// TIA Portal project "SistemaSupervisorio" (V17)
// Engenharia de Software 1

(* hardware
DEVICE "S7-1500/ET200MP station_1"  S7-1500 station
   slot 0: "RACK_CPU_1500"  Rack  6ES7 590-1***0-0AA0
   slot 1: "CPU_1500"  CPU 1511-1 PN  6ES7 511-1AK00-0AB0  V1.8
      slot 3: "CPU display_1"  6ES7591-1AA00-0AA0
      slot 32768: "PROFINET interface_1500"  X1
         slot 32769: "Port_1"  X1 P1
         slot 32770: "Port_2"  X1 P2
   slot 2: "DI1_1500"  DI 16x24VDC BA  6ES7 521-1BH10-0AA0  V1.1
   slot 3: "DO1_1500"  DQ 16x24VDC/0.5A BA  6ES7 522-1BH10-0AA0  V1.1
   slot 4: "AI/AO1_1500"  AI/AQ 4xU/I/RTD/TC / 2xU/I ST  6ES7 534-7QE00-0AB0  V1.0
*)

// ===== PLC "CPU_1500"  CPU 1511-1 PN =====

VAR_GLOBAL   // PLC tag table "Default tag table"
   "%I0.0" AT %I0.0 : Bool;   // I0.0 - Channel0 InDigitalCPU_1500
   "%I0.1" AT %I0.1 : Bool;   // I0.1 - Channel1 InDigitalCPU_1500
   "%I0.2" AT %I0.2 : Bool;   // I0.2 - Channel2 InDigitalCPU_1500
   "%I0.3" AT %I0.3 : Bool;   // I0.3 - Channel3 InDigitalCPU_1500
   "%I0.4" AT %I0.4 : Bool;   // I0.4 - Channel4 InDigitalCPU_1500
   "%I0.5" AT %I0.5 : Bool;   // I0.5 - Channel5 InDigitalCPU_1500
   "%I0.6" AT %I0.6 : Bool;   // I0.6 - Channel6 InDigitalCPU_1500
   "%I0.7" AT %I0.7 : Bool;   // I0.7 - Channel7 InDigitalCPU_1500
   "%I1.0" AT %I1.0 : Bool;   // I1.0 - Channel10 InDigitalCPU_1500
   "%I1.1" AT %I1.1 : Bool;   // I1.1 - Channel11 InDigitalCPU_1500
   "%I1.2" AT %I1.2 : Bool;   // I1.2 - Channel12 InDigitalCPU_1500
   "%I1.3" AT %I1.3 : Bool;   // I1.3 - Channel13 InDigitalCPU_1500
   "%I1.4" AT %I1.4 : Bool;   // I1.4 - Channel14 InDigitalCPU_1500
   "%I1.5" AT %I1.5 : Bool;   // I1.5 - Channel15 InDigitalCPU_1500
   "%I1.6" AT %I1.6 : Bool;   // I1.6 - Channel16 InDigitalCPU_1500
   "%I1.7" AT %I1.7 : Bool;   // I1.7 - Channel17 InDigitalCPU_1500
   "%IW2" AT %IW2 : Int;   // IW2 - Channel0 InAnalogAI/AO_1500
   "%IW4" AT %IW4 : Int;   // IW4 - Channel1 InAnalogAI/AO_1500
   "%IW6" AT %IW6 : Int;   // IW6 - Channel3 InAnalogAI/AO_1500
   "%IW8" AT %IW8 : Int;   // IW8 - Channel4 InAnalogAI/AO_1500
   "%QW2" AT %QW2 : Int;   // %QW2 - Channel0 OutAnalogAI/AO_1500
   "%QW4" AT %QW4 : Int;   // %QW4 - Channel1 OutAnalogAI/AO_1500
   "%Q0.0" AT %Q0.0 : Bool;   // Q0.0 - Channel0 OutDigitalDO_1500
   "%Q0.1" AT %Q0.1 : Bool;   // Q0.1 - Channel1 OutDigitalDO_1500
   "%Q0.2" AT %Q0.2 : Bool;   // Q1.0 - Channel2 OutDigitalDO_1500
   "%Q0.3" AT %Q0.3 : Bool;   // Q0.3 - Channel3 OutDigitalDO_1500
   "%Q0.4" AT %Q0.4 : Bool;   // Q0.4 - Channel4 OutDigitalDO_1500
   "%Q0.5" AT %Q0.5 : Bool;   // Q0.5 - Channel5 OutDigitalDO_1500
   "%Q0.6" AT %Q0.6 : Bool;   // Q0.6 - Channel6 OutDigitalDO_1500
   "%Q0.7" AT %Q0.7 : Bool;   // Q0.7 - Channel7 OutDigitalDO_1500
   "%Q1.0" AT %Q1.0 : Bool;   // Q1.0 - Channel10 OutDigitalDO_1500
   "%Q1.1" AT %Q1.1 : Bool;   // Q1.1 - Channel11 OutDigitalDO_1500
   "%Q1.2" AT %Q1.2 : Bool;   // Q1.2 - Channel12 OutDigitalDO_1500
   "%Q1.3" AT %Q1.3 : Bool;   // Q1.3 - Channel13 OutDigitalDO_1500
   "%Q1.4" AT %Q1.4 : Bool;   // Q1.4 - Channel14 OutDigitalDO_1500
   "%Q1.5" AT %Q1.5 : Bool;   // Q1.5 - Channel15 OutDigitalDO_1500
   "%Q1.6" AT %Q1.6 : Bool;   // Q1.6 - Channel16 OutDigitalDO_1500
   "%Q1.7" AT %Q1.7 : Bool;   // Q1.7 - Channel17 OutDigitalDO_1500
   "System_Byte" AT %MB100 : Byte;
   "FirstScan" AT %M100.0 : Bool;
   "DiagStatusUpdate" AT %M100.1 : Bool;
   "AlwaysTRUE" AT %M100.2 : Bool;
   "AlwaysFALSE" AT %M100.3 : Bool;
   "Tag_1" AT %M150.1 : Bool;
END_VAR

// folder: 001 - IOs/DBs

DATA_BLOCK "Ed"   // DB1
{ S7_Optimized_Access := 'FALSE' }
VERSION : 0.1
   VAR
      "I0.0" : Bool;   // I0.0 - Channel0 InDigitalCPU_ENG1
      "I0.1" : Bool;   // I0.1 - Channel1 InDigitalCPU_ENG1
      "I0.2" : Bool;   // I0.2 - Channel2 InDigitalCPU_ENG1
      "I0.3" : Bool;   // I0.3 - Channel3 InDigitalCPU_ENG1
      "I0.4" : Bool;   // I0.4 - Channel4 InDigitalCPU_ENG1
      "I0.5" : Bool;   // I0.5 - Channel5 InDigitalCPU_ENG1
      "I0.6" : Bool;   // I0.6 - Channel6 InDigitalCPU_ENG1
      "I0.7" : Bool;   // I0.7 - Channel7 InDigitalCPU_ENG1
      "I1.0" : Bool;   // I1.0 - Channel8 InDigitalCPU_ENG1
      "I1.1" : Bool;   // I1.1 - Channel9 InDigitalCPU_ENG1
      "I1.2" : Bool;   // I1.2 - Channel10, InDigitalCPU_ENG1
      "I1.3" : Bool;   // I1.3 - Channel11 InDigitalCPU_ENG1
      "I1.4" : Bool;   // I1.4 - Channel12 InDigitalCPU_ENG1
      "I1.5" : Bool;   // I1.5 - Channel13 InDigitalCPU_ENG1
      "I1.6" : Bool;
      "I1.7" : Bool;
      Simulation : Struct
         Ed : Struct
            "I0.0" : Bool;
            "I0.1" : Bool;
            "I0.2" : Bool;
            "I0.3" : Bool;
            "I0.4" : Bool;
            "I0.5" : Bool;
            "I0.6" : Bool;
            "I0.7" : Bool;
            "I1.0" : Bool;
            "I1.1" : Bool;
            "I1.2" : Bool;
            "I1.3" : Bool;
            "I1.4" : Bool;
            "I1.5" : Bool;
            "I1.6" : Bool;
            "I1.7" : Bool;
         END_STRUCT;
         Test : Struct
            "I0.0" : Bool;
            "I0.1" : Bool;
            "I0.2" : Bool;
            "I0.3" : Bool;
            "I0.4" : Bool;
            "I0.5" : Bool;
            "I0.6" : Bool;
            "I0.7" : Bool;
            "I1.0" : Bool;
            "I1.1" : Bool;
            "I1.2" : Bool;
            "I1.3" : Bool;
            "I1.4" : Bool;
            "I1.5" : Bool;
            "I1.6" : Bool;
            "I1.7" : Bool;
            All : Bool;
         END_STRUCT;
         Enable : Struct
            "I0.0" : Bool;
            "I0.1" : Bool;
            "I0.2" : Bool;
            "I0.3" : Bool;
            "I0.4" : Bool;
            "I0.5" : Bool;
            "I0.6" : Bool;
            "I0.7" : Bool;
            "I1.0" : Bool;
            "I1.1" : Bool;
            "I1.2" : Bool;
            "I1.3" : Bool;
            "I1.4" : Bool;
            "I1.5" : Bool;
            "I1.6" : Bool;
            "I1.7" : Bool;
            All : Bool;
         END_STRUCT;
      END_STRUCT;
   END_VAR
BEGIN
END_DATA_BLOCK

DATA_BLOCK "Sd"   // DB2
{ S7_Optimized_Access := 'FALSE' }
VERSION : 0.1
   VAR
      "Q0.0" : Bool;   // Q0.0 - Channel0 OutDigitalCPU_ENG1
      "Q0.1" : Bool;   // Q0.1 - Channel1 OutDigitalCPU_ENG1
      "Q0.2" : Bool;   // Q0.2 - Channel2 OutDigitalCPU_ENG1
      "Q0.3" : Bool;   // Q0.3 - Channel3 OutDigitalCPU_ENG1
      "Q0.4" : Bool;   // Q0.4 - Channel4 OutDigitalCPU_ENG1
      "Q0.5" : Bool;   // Q0.5 - Channel5 OutDigitalCPU_ENG1
      "Q0.6" : Bool;   // Q0.6 - Channel6 OutDigitalCPU_ENG1
      "Q0.7" : Bool;   // Q0.7 - Channel7 OutDigitalCPU_ENG1
      "Q1.0" : Bool;   // Q1.1 - Channel8 OutDigitalCPU_ENG1
      "Q1.1" : Bool;   // Q1.2 - Channel9 OutDigitalCPU_ENG1
      "Q1.2" : Bool;
      "Q1.3" : Bool;
      "Q1.4" : Bool;
      "Q1.5" : Bool;
      "Q1.6" : Bool;
      "Q1.7" : Bool;
      Simulation : Struct
         Sd : Struct
            "Q0.0" : Bool;   // Q0.0 - Channel0 OutDigitalCPU_ENG1
            "Q0.1" : Bool;   // Q0.1 - Channel1 OutDigitalCPU_ENG1
            "Q0.2" : Bool;   // Q0.2 - Channel2 OutDigitalCPU_ENG1
            "Q0.3" : Bool;   // Q0.3 - Channel3 OutDigitalCPU_ENG1
            "Q0.4" : Bool;   // Q0.4 - Channel4 OutDigitalCPU_ENG1
            "Q0.5" : Bool;   // Q0.5 - Channel5 OutDigitalCPU_ENG1
            "Q0.6" : Bool;   // Q0.6 - Channel6 OutDigitalCPU_ENG1
            "Q0.7" : Bool;   // Q0.7 - Channel7 OutDigitalCPU_ENG1
            "Q1.0" : Bool;   // Q1.1 - Channel8 OutDigitalCPU_ENG1
            "Q1.1" : Bool;   // Q1.2 - Channel9 OutDigitalCPU_ENG1
            "Q1.2" : Bool;
            "Q1.3" : Bool;
            "Q1.4" : Bool;
            "Q1.5" : Bool;
            "Q1.6" : Bool;
            "Q1.7" : Bool;
         END_STRUCT;
         Test : Struct
            "Q0.0" : Bool;
            "Q0.1" : Bool;
            "Q0.2" : Bool;
            "Q0.3" : Bool;
            "Q0.4" : Bool;
            "Q0.5" : Bool;
            "Q0.6" : Bool;
            "Q0.7" : Bool;
            "Q1.0" : Bool;
            "Q1.1" : Bool;
            "Q1.2" : Bool;
            "Q1.3" : Bool;
            "Q1.4" : Bool;
            "Q1.5" : Bool;
            "Q1.6" : Bool;
            "Q1.7" : Bool;
            All : Bool;
         END_STRUCT;
         Enable : Struct
            "Q0.0" : Bool;
            "Q0.1" : Bool;
            "Q0.2" : Bool;
            "Q0.3" : Bool;
            "Q0.4" : Bool;
            "Q0.5" : Bool;
            "Q0.6" : Bool;
            "Q0.7" : Bool;
            "Q1.0" : Bool;
            "Q1.1" : Bool;
            "Q1.2" : Bool;
            "Q1.3" : Bool;
            "Q1.4" : Bool;
            "Q1.5" : Bool;
            "Q1.6" : Bool;
            "Q1.7" : Bool;
            All : Bool;
         END_STRUCT;
      END_STRUCT;
   END_VAR
BEGIN
END_DATA_BLOCK

DATA_BLOCK "Ea"   // DB3
{ S7_Optimized_Access := 'FALSE' }
VERSION : 0.1
   VAR
      IW2 : Int;   // IW64 - Channel0 InAnalogCPU_ENG1
      IW4 : Int;   // IW66 - Channel1 InAnalogCPU_ENG1
      IW6 : Int;   // IW96 - Channel0 InAnalogAI/AO_ENG1
      IW8 : Int;   // IW98 - Channel1 InAnalogAI/AO_ENG1
      Simulation : Struct
         Ea : Struct
            IW2 : Int;   // IW64 - Channel0 InAnalogCPU_ENG1
            IW4 : Int;   // IW66 - Channel1 InAnalogCPU_ENG1
            IW6 : Int;   // IW96 - Channel0 InAnalogAI/AO_ENG1
            IW8 : Int;   // IW98 - Channel1 InAnalogAI/AO_ENG1
         END_STRUCT;
         Test : Struct
            IW2 : DInt;   // IW64 - Channel0 InAnalogCPU_ENG1
            IW4 : DInt;   // IW66 - Channel1 InAnalogCPU_ENG1
            IW6 : DInt;   // IW96 - Channel0 InAnalogAI/AO_ENG1
            IW8 : DInt;   // IW98 - Channel1 InAnalogAI/AO_ENG1
            All : DInt;
         END_STRUCT;
         Enable : Struct
            IW2 : Bool;   // IW64 - Channel0 InAnalogCPU_ENG1
            IW4 : Bool;   // IW66 - Channel1 InAnalogCPU_ENG1
            IW6 : Bool;   // IW96 - Channel0 InAnalogAI/AO_ENG1
            IW8 : Bool;   // IW98 - Channel1 InAnalogAI/AO_ENG1
            All : Bool;
         END_STRUCT;
      END_STRUCT;
   END_VAR
BEGIN
END_DATA_BLOCK

DATA_BLOCK "Sa"   // DB4
{ S7_Optimized_Access := 'FALSE' }
VERSION : 0.1
   VAR
      QW2 : Int;   // IW96 - Channel0 OutAnalogCPU_AI/AO
      QW4 : Int;   // IW98 - Channel1 OutAnalogCPU_AI/AO
      Simulation : Struct
         Sa : Struct
            QW2 : Int;
            QW4 : Int;
         END_STRUCT;
         Test : Struct
            QW2 : DInt;
            QW4 : DInt;
            All : DInt;
         END_STRUCT;
         Enable : Struct
            QW2 : Bool;
            QW4 : Bool;
            All : Bool;
         END_STRUCT;
      END_STRUCT;
   END_VAR
BEGIN
END_DATA_BLOCK

// folder: 002 - Comunication Node-Red/DBs

DATA_BLOCK "Node-Red"   // DB6
{ S7_Optimized_Access := 'FALSE' }
VERSION : 0.1
   VAR
      escreveNodeRedBool : Bool;
      escreveNodeRedDint : DInt;
      recebeNodeRedBool : Bool;
      recebeNodeRedReal : Real;
      auxEscreveNodRedReal : DInt;
      auxRecebeNodeRedReal : DInt;
      statusMaquinaNodeRed : Int;
      "enviaStatusNode-Red" : Int;
      avisosMaquinaNodeRed : Int;
      enviaAvisosMaquinaNodeRed : Int;
      "alarmesNode-Red" : Int;
      enviaAlarmesNodeRed : Int;
      "valorVelocidadeNode-Red" : Int;
      "enviaValorVelocidadeNode-Red" : Int;
      valorProducao : Int;
      enviaValorProducao : Int;
      enableEnviaValorProdução : Bool;
      enableEnviaValorVelocidade : Bool;
   END_VAR
BEGIN
END_DATA_BLOCK

// folder: 100 - DBs

DATA_BLOCK "x"   // DB5
{ S7_Optimized_Access := 'TRUE' }
VERSION : 0.1
   VAR RETAIN
      Constantes : Struct
         "+int" : Int := 32767;
         "-int" : Int := -32767;
         "0int" : Int := 0;
      END_STRUCT;
      AlwaysFalse : Bool := 0;
      AlwaysTrue : Bool := 1;
   END_VAR
   VAR
      Timers : Struct
         t1s : Bool;
         t5s : Bool;
         t10s : Bool;
      END_STRUCT;
   END_VAR
BEGIN
END_DATA_BLOCK

// folder: System blocks/Program resources

DATA_BLOCK "tonTimer5seg"   // DB7
{ S7_Optimized_Access := 'TRUE' }
AUTHOR : Simatic
FAMILY : IEC
NAME : IEC_TMR
VERSION : 1.0
// stored: InstanceOfName IEC_TIMER
"IEC_TIMER"
BEGIN
END_DATA_BLOCK

DATA_BLOCK "tonTimer10seg"   // DB8
{ S7_Optimized_Access := 'TRUE' }
AUTHOR : Simatic
FAMILY : IEC
NAME : IEC_TMR
VERSION : 1.0
// stored: InstanceOfName IEC_TIMER
"IEC_TIMER"
BEGIN
END_DATA_BLOCK

DATA_BLOCK "tonTimer1seg"   // DB9
{ S7_Optimized_Access := 'TRUE' }
AUTHOR : Simatic
FAMILY : IEC
NAME : IEC_TMR
VERSION : 1.0
// stored: InstanceOfName IEC_TIMER
"IEC_TIMER"
BEGIN
END_DATA_BLOCK

// folder: (top level)

ORGANIZATION_BLOCK "Main"   // OB1, LAD, ProgramCycle
TITLE = "Main Program Sweep (Cycle)"
{ S7_Optimized_Access := 'TRUE' }
VERSION : 0.1
   VAR_INPUT
      Initial_Call : Bool;   // Initial call of this OB
      Remanence : Bool;   // =True, if remanent data are available
   END_VAR
BEGIN

REGION Network 1: 01 - Digital Inputs
   // 01 - Digital Input
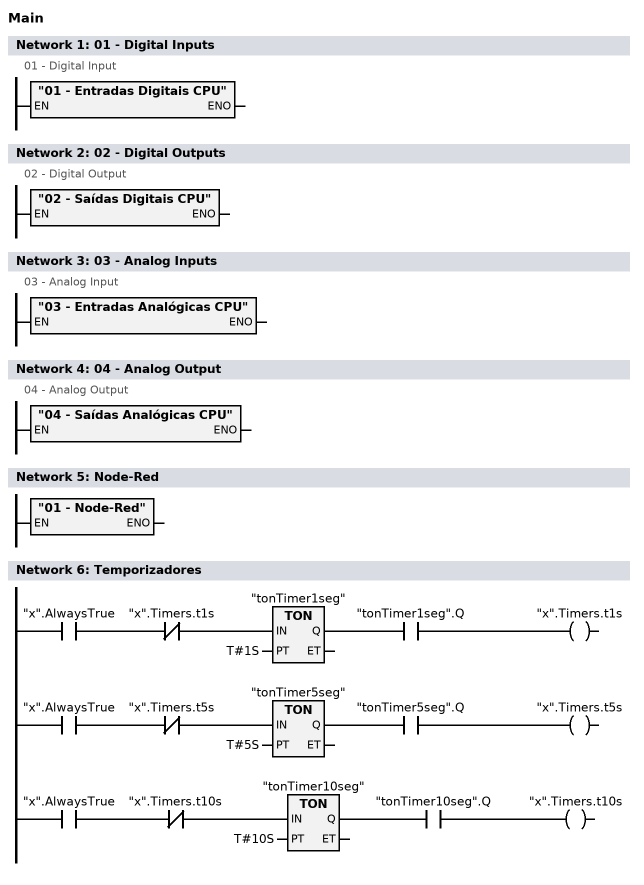
   RUNG wire#powerrail
      "01 - Entradas Digitais CPU"()
   END_RUNG
   // the same network as SCL:
   "01 - Entradas Digitais CPU"();
END_REGION

REGION Network 2: 02 - Digital Outputs
   // 02 - Digital Output
   RUNG wire#powerrail
      "02 - Saídas Digitais CPU"()
   END_RUNG
   // the same network as SCL:
   "02 - Saídas Digitais CPU"();
END_REGION

REGION Network 3: 03 - Analog Inputs
   // 03 - Analog Input
   RUNG wire#powerrail
      "03 - Entradas Analógicas CPU"()
   END_RUNG
   // the same network as SCL:
   "03 - Entradas Analógicas CPU"();
END_REGION

REGION Network 4: 04 - Analog Output
   // 04 - Analog Output
   RUNG wire#powerrail
      "04 - Saídas Analógicas CPU"()
   END_RUNG
   // the same network as SCL:
   "04 - Saídas Analógicas CPU"();
END_REGION

REGION Network 5: Node-Red
   RUNG wire#powerrail
      "01 - Node-Red"()
   END_RUNG
   // the same network as SCL:
   "01 - Node-Red"();
END_REGION

REGION Network 6: Temporizadores
   "tonTimer1seg".TON(IN := "x".AlwaysTrue AND NOT "x".Timers.t1s, PT := T#1S);
   "x".Timers.t1s := "tonTimer1seg".Q AND "tonTimer1seg".Q;
   "tonTimer5seg".TON(IN := "x".AlwaysTrue AND NOT "x".Timers.t5s, PT := T#5S);
   "x".Timers.t5s := "tonTimer5seg".Q AND "tonTimer5seg".Q;
   "tonTimer10seg".TON(IN := "x".AlwaysTrue AND NOT "x".Timers.t10s, PT := T#10S);
   "x".Timers.t10s := "tonTimer10seg".Q AND "tonTimer10seg".Q;
END_REGION
END_ORGANIZATION_BLOCK

// folder: 001 - IOs

FUNCTION "01 - Entradas Digitais CPU" : Void   // FC1, LAD
TITLE = 01 - Digital Inputs
{ S7_Optimized_Access := 'TRUE' }
VERSION : 0.1
// 01 - Digital Inputs
   VAR_TEMP
      testeAllHabilitado : Bool;
      testeAllDesabilitado : Bool;
   END_VAR
BEGIN

REGION Network 1: 00 - Digital Input %I0.0
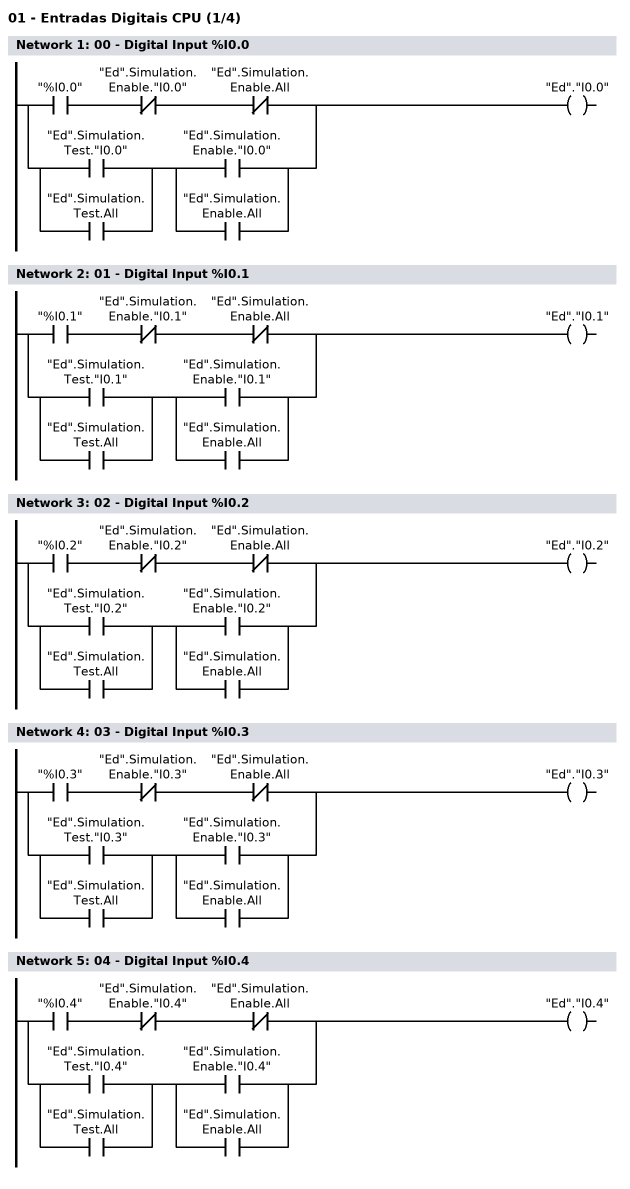
   RUNG wire#powerrail
      Contact( "%I0.0" )
      I_Contact( "Ed".Simulation.Enable."I0.0" )
      I_Contact( "Ed".Simulation.Enable.All )
      wire#w1
      Coil( "Ed"."I0.0" )
   END_RUNG
   RUNG wire#powerrail
      Contact( "Ed".Simulation.Test."I0.0" )
      wire#w2
      Contact( "Ed".Simulation.Enable."I0.0" )
   END_RUNG wire#w1
   RUNG wire#powerrail
      Contact( "Ed".Simulation.Test.All )
   END_RUNG wire#w2
   RUNG wire#w2
      Contact( "Ed".Simulation.Enable.All )
   END_RUNG wire#w1
   // the same network as SCL:
   "Ed"."I0.0" := ("%I0.0" AND NOT "Ed".Simulation.Enable."I0.0" AND NOT "Ed".Simulation.Enable.All) OR (("Ed".Simulation.Test."I0.0" OR "Ed".Simulation.Test.All) AND ("Ed".Simulation.Enable."I0.0" OR "Ed".Simulation.Enable.All));
END_REGION

REGION Network 2: 01 - Digital Input %I0.1
   RUNG wire#powerrail
      Contact( "%I0.1" )
      I_Contact( "Ed".Simulation.Enable."I0.1" )
      I_Contact( "Ed".Simulation.Enable.All )
      wire#w1
      Coil( "Ed"."I0.1" )
   END_RUNG
   RUNG wire#powerrail
      Contact( "Ed".Simulation.Test."I0.1" )
      wire#w2
      Contact( "Ed".Simulation.Enable."I0.1" )
   END_RUNG wire#w1
   RUNG wire#powerrail
      Contact( "Ed".Simulation.Test.All )
   END_RUNG wire#w2
   RUNG wire#w2
      Contact( "Ed".Simulation.Enable.All )
   END_RUNG wire#w1
   // the same network as SCL:
   "Ed"."I0.1" := ("%I0.1" AND NOT "Ed".Simulation.Enable."I0.1" AND NOT "Ed".Simulation.Enable.All) OR (("Ed".Simulation.Test."I0.1" OR "Ed".Simulation.Test.All) AND ("Ed".Simulation.Enable."I0.1" OR "Ed".Simulation.Enable.All));
END_REGION

REGION Network 3: 02 - Digital Input %I0.2
   RUNG wire#powerrail
      Contact( "%I0.2" )
      I_Contact( "Ed".Simulation.Enable."I0.2" )
      I_Contact( "Ed".Simulation.Enable.All )
      wire#w1
      Coil( "Ed"."I0.2" )
   END_RUNG
   RUNG wire#powerrail
      Contact( "Ed".Simulation.Test."I0.2" )
      wire#w2
      Contact( "Ed".Simulation.Enable."I0.2" )
   END_RUNG wire#w1
   RUNG wire#powerrail
      Contact( "Ed".Simulation.Test.All )
   END_RUNG wire#w2
   RUNG wire#w2
      Contact( "Ed".Simulation.Enable.All )
   END_RUNG wire#w1
   // the same network as SCL:
   "Ed"."I0.2" := ("%I0.2" AND NOT "Ed".Simulation.Enable."I0.2" AND NOT "Ed".Simulation.Enable.All) OR (("Ed".Simulation.Test."I0.2" OR "Ed".Simulation.Test.All) AND ("Ed".Simulation.Enable."I0.2" OR "Ed".Simulation.Enable.All));
END_REGION

REGION Network 4: 03 - Digital Input %I0.3
   RUNG wire#powerrail
      Contact( "%I0.3" )
      I_Contact( "Ed".Simulation.Enable."I0.3" )
      I_Contact( "Ed".Simulation.Enable.All )
      wire#w1
      Coil( "Ed"."I0.3" )
   END_RUNG
   RUNG wire#powerrail
      Contact( "Ed".Simulation.Test."I0.3" )
      wire#w2
      Contact( "Ed".Simulation.Enable."I0.3" )
   END_RUNG wire#w1
   RUNG wire#powerrail
      Contact( "Ed".Simulation.Test.All )
   END_RUNG wire#w2
   RUNG wire#w2
      Contact( "Ed".Simulation.Enable.All )
   END_RUNG wire#w1
   // the same network as SCL:
   "Ed"."I0.3" := ("%I0.3" AND NOT "Ed".Simulation.Enable."I0.3" AND NOT "Ed".Simulation.Enable.All) OR (("Ed".Simulation.Test."I0.3" OR "Ed".Simulation.Test.All) AND ("Ed".Simulation.Enable."I0.3" OR "Ed".Simulation.Enable.All));
END_REGION

REGION Network 5: 04 - Digital Input %I0.4
   RUNG wire#powerrail
      Contact( "%I0.4" )
      I_Contact( "Ed".Simulation.Enable."I0.4" )
      I_Contact( "Ed".Simulation.Enable.All )
      wire#w1
      Coil( "Ed"."I0.4" )
   END_RUNG
   RUNG wire#powerrail
      Contact( "Ed".Simulation.Test."I0.4" )
      wire#w2
      Contact( "Ed".Simulation.Enable."I0.4" )
   END_RUNG wire#w1
   RUNG wire#powerrail
      Contact( "Ed".Simulation.Test.All )
   END_RUNG wire#w2
   RUNG wire#w2
      Contact( "Ed".Simulation.Enable.All )
   END_RUNG wire#w1
   // the same network as SCL:
   "Ed"."I0.4" := ("%I0.4" AND NOT "Ed".Simulation.Enable."I0.4" AND NOT "Ed".Simulation.Enable.All) OR (("Ed".Simulation.Test."I0.4" OR "Ed".Simulation.Test.All) AND ("Ed".Simulation.Enable."I0.4" OR "Ed".Simulation.Enable.All));
END_REGION

REGION Network 6: 05 - Digital Input %I0.5
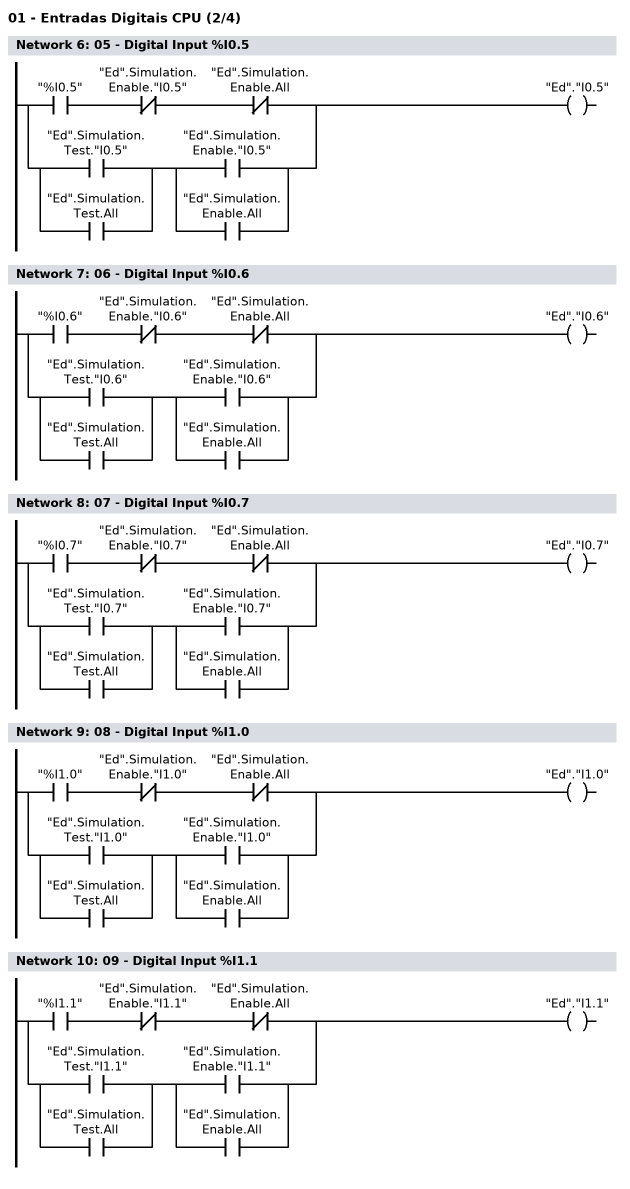
   RUNG wire#powerrail
      Contact( "%I0.5" )
      I_Contact( "Ed".Simulation.Enable."I0.5" )
      I_Contact( "Ed".Simulation.Enable.All )
      wire#w1
      Coil( "Ed"."I0.5" )
   END_RUNG
   RUNG wire#powerrail
      Contact( "Ed".Simulation.Test."I0.5" )
      wire#w2
      Contact( "Ed".Simulation.Enable."I0.5" )
   END_RUNG wire#w1
   RUNG wire#powerrail
      Contact( "Ed".Simulation.Test.All )
   END_RUNG wire#w2
   RUNG wire#w2
      Contact( "Ed".Simulation.Enable.All )
   END_RUNG wire#w1
   // the same network as SCL:
   "Ed"."I0.5" := ("%I0.5" AND NOT "Ed".Simulation.Enable."I0.5" AND NOT "Ed".Simulation.Enable.All) OR (("Ed".Simulation.Test."I0.5" OR "Ed".Simulation.Test.All) AND ("Ed".Simulation.Enable."I0.5" OR "Ed".Simulation.Enable.All));
END_REGION

REGION Network 7: 06 - Digital Input %I0.6
   RUNG wire#powerrail
      Contact( "%I0.6" )
      I_Contact( "Ed".Simulation.Enable."I0.6" )
      I_Contact( "Ed".Simulation.Enable.All )
      wire#w1
      Coil( "Ed"."I0.6" )
   END_RUNG
   RUNG wire#powerrail
      Contact( "Ed".Simulation.Test."I0.6" )
      wire#w2
      Contact( "Ed".Simulation.Enable."I0.6" )
   END_RUNG wire#w1
   RUNG wire#powerrail
      Contact( "Ed".Simulation.Test.All )
   END_RUNG wire#w2
   RUNG wire#w2
      Contact( "Ed".Simulation.Enable.All )
   END_RUNG wire#w1
   // the same network as SCL:
   "Ed"."I0.6" := ("%I0.6" AND NOT "Ed".Simulation.Enable."I0.6" AND NOT "Ed".Simulation.Enable.All) OR (("Ed".Simulation.Test."I0.6" OR "Ed".Simulation.Test.All) AND ("Ed".Simulation.Enable."I0.6" OR "Ed".Simulation.Enable.All));
END_REGION

REGION Network 8: 07 - Digital Input %I0.7
   RUNG wire#powerrail
      Contact( "%I0.7" )
      I_Contact( "Ed".Simulation.Enable."I0.7" )
      I_Contact( "Ed".Simulation.Enable.All )
      wire#w1
      Coil( "Ed"."I0.7" )
   END_RUNG
   RUNG wire#powerrail
      Contact( "Ed".Simulation.Test."I0.7" )
      wire#w2
      Contact( "Ed".Simulation.Enable."I0.7" )
   END_RUNG wire#w1
   RUNG wire#powerrail
      Contact( "Ed".Simulation.Test.All )
   END_RUNG wire#w2
   RUNG wire#w2
      Contact( "Ed".Simulation.Enable.All )
   END_RUNG wire#w1
   // the same network as SCL:
   "Ed"."I0.7" := ("%I0.7" AND NOT "Ed".Simulation.Enable."I0.7" AND NOT "Ed".Simulation.Enable.All) OR (("Ed".Simulation.Test."I0.7" OR "Ed".Simulation.Test.All) AND ("Ed".Simulation.Enable."I0.7" OR "Ed".Simulation.Enable.All));
END_REGION

REGION Network 9: 08 - Digital Input %I1.0
   RUNG wire#powerrail
      Contact( "%I1.0" )
      I_Contact( "Ed".Simulation.Enable."I1.0" )
      I_Contact( "Ed".Simulation.Enable.All )
      wire#w1
      Coil( "Ed"."I1.0" )
   END_RUNG
   RUNG wire#powerrail
      Contact( "Ed".Simulation.Test."I1.0" )
      wire#w2
      Contact( "Ed".Simulation.Enable."I1.0" )
   END_RUNG wire#w1
   RUNG wire#powerrail
      Contact( "Ed".Simulation.Test.All )
   END_RUNG wire#w2
   RUNG wire#w2
      Contact( "Ed".Simulation.Enable.All )
   END_RUNG wire#w1
   // the same network as SCL:
   "Ed"."I1.0" := ("%I1.0" AND NOT "Ed".Simulation.Enable."I1.0" AND NOT "Ed".Simulation.Enable.All) OR (("Ed".Simulation.Test."I1.0" OR "Ed".Simulation.Test.All) AND ("Ed".Simulation.Enable."I1.0" OR "Ed".Simulation.Enable.All));
END_REGION

REGION Network 10: 09 - Digital Input %I1.1
   RUNG wire#powerrail
      Contact( "%I1.1" )
      I_Contact( "Ed".Simulation.Enable."I1.1" )
      I_Contact( "Ed".Simulation.Enable.All )
      wire#w1
      Coil( "Ed"."I1.1" )
   END_RUNG
   RUNG wire#powerrail
      Contact( "Ed".Simulation.Test."I1.1" )
      wire#w2
      Contact( "Ed".Simulation.Enable."I1.1" )
   END_RUNG wire#w1
   RUNG wire#powerrail
      Contact( "Ed".Simulation.Test.All )
   END_RUNG wire#w2
   RUNG wire#w2
      Contact( "Ed".Simulation.Enable.All )
   END_RUNG wire#w1
   // the same network as SCL:
   "Ed"."I1.1" := ("%I1.1" AND NOT "Ed".Simulation.Enable."I1.1" AND NOT "Ed".Simulation.Enable.All) OR (("Ed".Simulation.Test."I1.1" OR "Ed".Simulation.Test.All) AND ("Ed".Simulation.Enable."I1.1" OR "Ed".Simulation.Enable.All));
END_REGION

REGION Network 11: 10 - Digital Input %I1.2
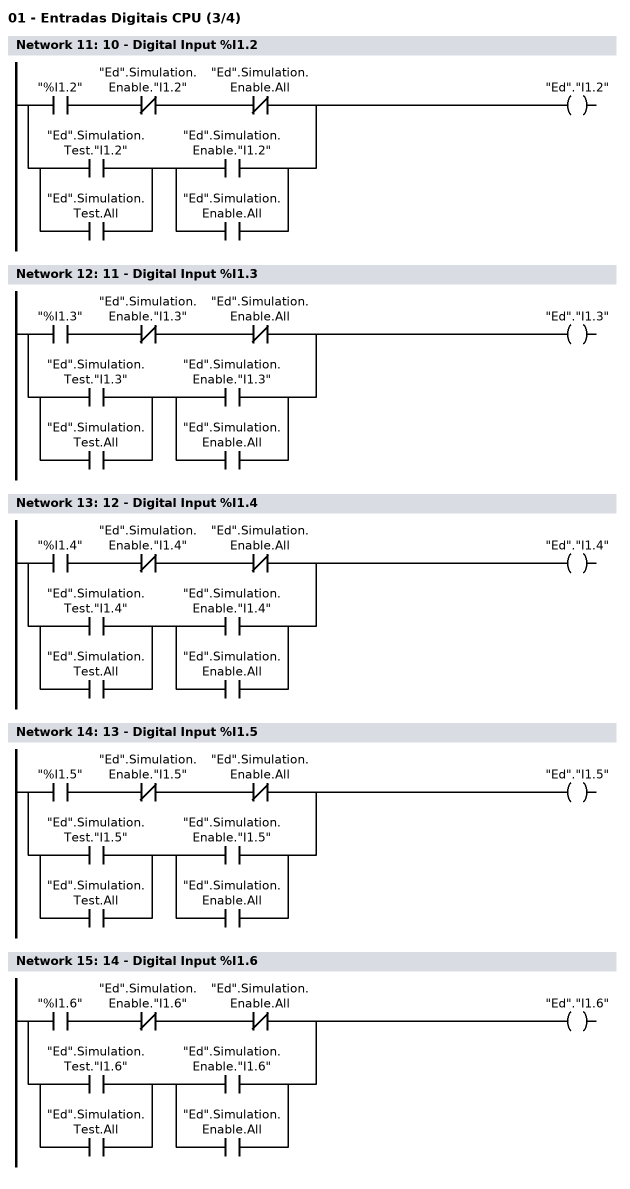
   RUNG wire#powerrail
      Contact( "%I1.2" )
      I_Contact( "Ed".Simulation.Enable."I1.2" )
      I_Contact( "Ed".Simulation.Enable.All )
      wire#w1
      Coil( "Ed"."I1.2" )
   END_RUNG
   RUNG wire#powerrail
      Contact( "Ed".Simulation.Test."I1.2" )
      wire#w2
      Contact( "Ed".Simulation.Enable."I1.2" )
   END_RUNG wire#w1
   RUNG wire#powerrail
      Contact( "Ed".Simulation.Test.All )
   END_RUNG wire#w2
   RUNG wire#w2
      Contact( "Ed".Simulation.Enable.All )
   END_RUNG wire#w1
   // the same network as SCL:
   "Ed"."I1.2" := ("%I1.2" AND NOT "Ed".Simulation.Enable."I1.2" AND NOT "Ed".Simulation.Enable.All) OR (("Ed".Simulation.Test."I1.2" OR "Ed".Simulation.Test.All) AND ("Ed".Simulation.Enable."I1.2" OR "Ed".Simulation.Enable.All));
END_REGION

REGION Network 12: 11 - Digital Input %I1.3
   RUNG wire#powerrail
      Contact( "%I1.3" )
      I_Contact( "Ed".Simulation.Enable."I1.3" )
      I_Contact( "Ed".Simulation.Enable.All )
      wire#w1
      Coil( "Ed"."I1.3" )
   END_RUNG
   RUNG wire#powerrail
      Contact( "Ed".Simulation.Test."I1.3" )
      wire#w2
      Contact( "Ed".Simulation.Enable."I1.3" )
   END_RUNG wire#w1
   RUNG wire#powerrail
      Contact( "Ed".Simulation.Test.All )
   END_RUNG wire#w2
   RUNG wire#w2
      Contact( "Ed".Simulation.Enable.All )
   END_RUNG wire#w1
   // the same network as SCL:
   "Ed"."I1.3" := ("%I1.3" AND NOT "Ed".Simulation.Enable."I1.3" AND NOT "Ed".Simulation.Enable.All) OR (("Ed".Simulation.Test."I1.3" OR "Ed".Simulation.Test.All) AND ("Ed".Simulation.Enable."I1.3" OR "Ed".Simulation.Enable.All));
END_REGION

REGION Network 13: 12 - Digital Input %I1.4
   RUNG wire#powerrail
      Contact( "%I1.4" )
      I_Contact( "Ed".Simulation.Enable."I1.4" )
      I_Contact( "Ed".Simulation.Enable.All )
      wire#w1
      Coil( "Ed"."I1.4" )
   END_RUNG
   RUNG wire#powerrail
      Contact( "Ed".Simulation.Test."I1.4" )
      wire#w2
      Contact( "Ed".Simulation.Enable."I1.4" )
   END_RUNG wire#w1
   RUNG wire#powerrail
      Contact( "Ed".Simulation.Test.All )
   END_RUNG wire#w2
   RUNG wire#w2
      Contact( "Ed".Simulation.Enable.All )
   END_RUNG wire#w1
   // the same network as SCL:
   "Ed"."I1.4" := ("%I1.4" AND NOT "Ed".Simulation.Enable."I1.4" AND NOT "Ed".Simulation.Enable.All) OR (("Ed".Simulation.Test."I1.4" OR "Ed".Simulation.Test.All) AND ("Ed".Simulation.Enable."I1.4" OR "Ed".Simulation.Enable.All));
END_REGION

REGION Network 14: 13 - Digital Input %I1.5
   RUNG wire#powerrail
      Contact( "%I1.5" )
      I_Contact( "Ed".Simulation.Enable."I1.5" )
      I_Contact( "Ed".Simulation.Enable.All )
      wire#w1
      Coil( "Ed"."I1.5" )
   END_RUNG
   RUNG wire#powerrail
      Contact( "Ed".Simulation.Test."I1.5" )
      wire#w2
      Contact( "Ed".Simulation.Enable."I1.5" )
   END_RUNG wire#w1
   RUNG wire#powerrail
      Contact( "Ed".Simulation.Test.All )
   END_RUNG wire#w2
   RUNG wire#w2
      Contact( "Ed".Simulation.Enable.All )
   END_RUNG wire#w1
   // the same network as SCL:
   "Ed"."I1.5" := ("%I1.5" AND NOT "Ed".Simulation.Enable."I1.5" AND NOT "Ed".Simulation.Enable.All) OR (("Ed".Simulation.Test."I1.5" OR "Ed".Simulation.Test.All) AND ("Ed".Simulation.Enable."I1.5" OR "Ed".Simulation.Enable.All));
END_REGION

REGION Network 15: 14 - Digital Input %I1.6
   RUNG wire#powerrail
      Contact( "%I1.6" )
      I_Contact( "Ed".Simulation.Enable."I1.6" )
      I_Contact( "Ed".Simulation.Enable.All )
      wire#w1
      Coil( "Ed"."I1.6" )
   END_RUNG
   RUNG wire#powerrail
      Contact( "Ed".Simulation.Test."I1.6" )
      wire#w2
      Contact( "Ed".Simulation.Enable."I1.6" )
   END_RUNG wire#w1
   RUNG wire#powerrail
      Contact( "Ed".Simulation.Test.All )
   END_RUNG wire#w2
   RUNG wire#w2
      Contact( "Ed".Simulation.Enable.All )
   END_RUNG wire#w1
   // the same network as SCL:
   "Ed"."I1.6" := ("%I1.6" AND NOT "Ed".Simulation.Enable."I1.6" AND NOT "Ed".Simulation.Enable.All) OR (("Ed".Simulation.Test."I1.6" OR "Ed".Simulation.Test.All) AND ("Ed".Simulation.Enable."I1.6" OR "Ed".Simulation.Enable.All));
END_REGION

REGION Network 16: 15 - Digital Input %I1.7
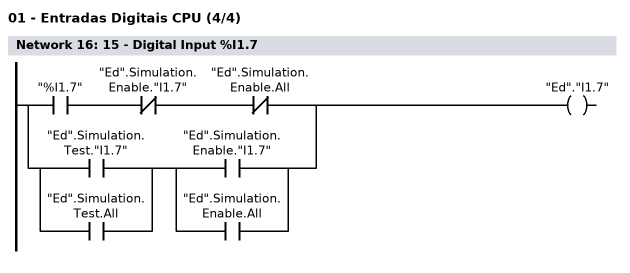
   RUNG wire#powerrail
      Contact( "%I1.7" )
      I_Contact( "Ed".Simulation.Enable."I1.7" )
      I_Contact( "Ed".Simulation.Enable.All )
      wire#w1
      Coil( "Ed"."I1.7" )
   END_RUNG
   RUNG wire#powerrail
      Contact( "Ed".Simulation.Test."I1.7" )
      wire#w2
      Contact( "Ed".Simulation.Enable."I1.7" )
   END_RUNG wire#w1
   RUNG wire#powerrail
      Contact( "Ed".Simulation.Test.All )
   END_RUNG wire#w2
   RUNG wire#w2
      Contact( "Ed".Simulation.Enable.All )
   END_RUNG wire#w1
   // the same network as SCL:
   "Ed"."I1.7" := ("%I1.7" AND NOT "Ed".Simulation.Enable."I1.7" AND NOT "Ed".Simulation.Enable.All) OR (("Ed".Simulation.Test."I1.7" OR "Ed".Simulation.Test.All) AND ("Ed".Simulation.Enable."I1.7" OR "Ed".Simulation.Enable.All));
END_REGION
END_FUNCTION

FUNCTION "02 - Saídas Digitais CPU" : Void   // FC2, LAD
TITLE = 01 - Digital Outputs
{ S7_Optimized_Access := 'TRUE' }
VERSION : 0.1
// 01 - Digital Outputs
BEGIN

REGION Network 1: 02 - Digital Output %Q0.0
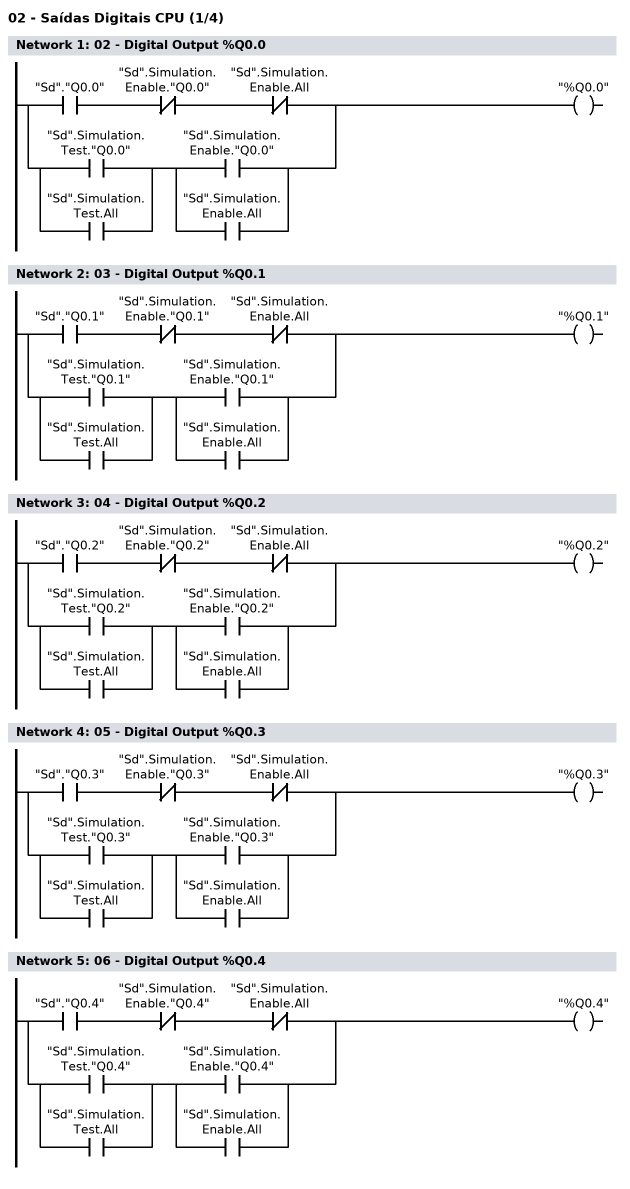
   RUNG wire#powerrail
      Contact( "Sd"."Q0.0" )
      I_Contact( "Sd".Simulation.Enable."Q0.0" )
      I_Contact( "Sd".Simulation.Enable.All )
      wire#w1
      Coil( "%Q0.0" )
   END_RUNG
   RUNG wire#powerrail
      Contact( "Sd".Simulation.Test."Q0.0" )
      wire#w2
      Contact( "Sd".Simulation.Enable."Q0.0" )
   END_RUNG wire#w1
   RUNG wire#powerrail
      Contact( "Sd".Simulation.Test.All )
   END_RUNG wire#w2
   RUNG wire#w2
      Contact( "Sd".Simulation.Enable.All )
   END_RUNG wire#w1
   // the same network as SCL:
   "%Q0.0" := ("Sd"."Q0.0" AND NOT "Sd".Simulation.Enable."Q0.0" AND NOT "Sd".Simulation.Enable.All) OR (("Sd".Simulation.Test."Q0.0" OR "Sd".Simulation.Test.All) AND ("Sd".Simulation.Enable."Q0.0" OR "Sd".Simulation.Enable.All));
END_REGION

REGION Network 2: 03 - Digital Output %Q0.1
   RUNG wire#powerrail
      Contact( "Sd"."Q0.1" )
      I_Contact( "Sd".Simulation.Enable."Q0.1" )
      I_Contact( "Sd".Simulation.Enable.All )
      wire#w1
      Coil( "%Q0.1" )
   END_RUNG
   RUNG wire#powerrail
      Contact( "Sd".Simulation.Test."Q0.1" )
      wire#w2
      Contact( "Sd".Simulation.Enable."Q0.1" )
   END_RUNG wire#w1
   RUNG wire#powerrail
      Contact( "Sd".Simulation.Test.All )
   END_RUNG wire#w2
   RUNG wire#w2
      Contact( "Sd".Simulation.Enable.All )
   END_RUNG wire#w1
   // the same network as SCL:
   "%Q0.1" := ("Sd"."Q0.1" AND NOT "Sd".Simulation.Enable."Q0.1" AND NOT "Sd".Simulation.Enable.All) OR (("Sd".Simulation.Test."Q0.1" OR "Sd".Simulation.Test.All) AND ("Sd".Simulation.Enable."Q0.1" OR "Sd".Simulation.Enable.All));
END_REGION

REGION Network 3: 04 - Digital Output %Q0.2
   RUNG wire#powerrail
      Contact( "Sd"."Q0.2" )
      I_Contact( "Sd".Simulation.Enable."Q0.2" )
      I_Contact( "Sd".Simulation.Enable.All )
      wire#w1
      Coil( "%Q0.2" )
   END_RUNG
   RUNG wire#powerrail
      Contact( "Sd".Simulation.Test."Q0.2" )
      wire#w2
      Contact( "Sd".Simulation.Enable."Q0.2" )
   END_RUNG wire#w1
   RUNG wire#powerrail
      Contact( "Sd".Simulation.Test.All )
   END_RUNG wire#w2
   RUNG wire#w2
      Contact( "Sd".Simulation.Enable.All )
   END_RUNG wire#w1
   // the same network as SCL:
   "%Q0.2" := ("Sd"."Q0.2" AND NOT "Sd".Simulation.Enable."Q0.2" AND NOT "Sd".Simulation.Enable.All) OR (("Sd".Simulation.Test."Q0.2" OR "Sd".Simulation.Test.All) AND ("Sd".Simulation.Enable."Q0.2" OR "Sd".Simulation.Enable.All));
END_REGION

REGION Network 4: 05 - Digital Output %Q0.3
   RUNG wire#powerrail
      Contact( "Sd"."Q0.3" )
      I_Contact( "Sd".Simulation.Enable."Q0.3" )
      I_Contact( "Sd".Simulation.Enable.All )
      wire#w1
      Coil( "%Q0.3" )
   END_RUNG
   RUNG wire#powerrail
      Contact( "Sd".Simulation.Test."Q0.3" )
      wire#w2
      Contact( "Sd".Simulation.Enable."Q0.3" )
   END_RUNG wire#w1
   RUNG wire#powerrail
      Contact( "Sd".Simulation.Test.All )
   END_RUNG wire#w2
   RUNG wire#w2
      Contact( "Sd".Simulation.Enable.All )
   END_RUNG wire#w1
   // the same network as SCL:
   "%Q0.3" := ("Sd"."Q0.3" AND NOT "Sd".Simulation.Enable."Q0.3" AND NOT "Sd".Simulation.Enable.All) OR (("Sd".Simulation.Test."Q0.3" OR "Sd".Simulation.Test.All) AND ("Sd".Simulation.Enable."Q0.3" OR "Sd".Simulation.Enable.All));
END_REGION

REGION Network 5: 06 - Digital Output %Q0.4
   RUNG wire#powerrail
      Contact( "Sd"."Q0.4" )
      I_Contact( "Sd".Simulation.Enable."Q0.4" )
      I_Contact( "Sd".Simulation.Enable.All )
      wire#w1
      Coil( "%Q0.4" )
   END_RUNG
   RUNG wire#powerrail
      Contact( "Sd".Simulation.Test."Q0.4" )
      wire#w2
      Contact( "Sd".Simulation.Enable."Q0.4" )
   END_RUNG wire#w1
   RUNG wire#powerrail
      Contact( "Sd".Simulation.Test.All )
   END_RUNG wire#w2
   RUNG wire#w2
      Contact( "Sd".Simulation.Enable.All )
   END_RUNG wire#w1
   // the same network as SCL:
   "%Q0.4" := ("Sd"."Q0.4" AND NOT "Sd".Simulation.Enable."Q0.4" AND NOT "Sd".Simulation.Enable.All) OR (("Sd".Simulation.Test."Q0.4" OR "Sd".Simulation.Test.All) AND ("Sd".Simulation.Enable."Q0.4" OR "Sd".Simulation.Enable.All));
END_REGION

REGION Network 6: 07 - Digital Output %Q0.5
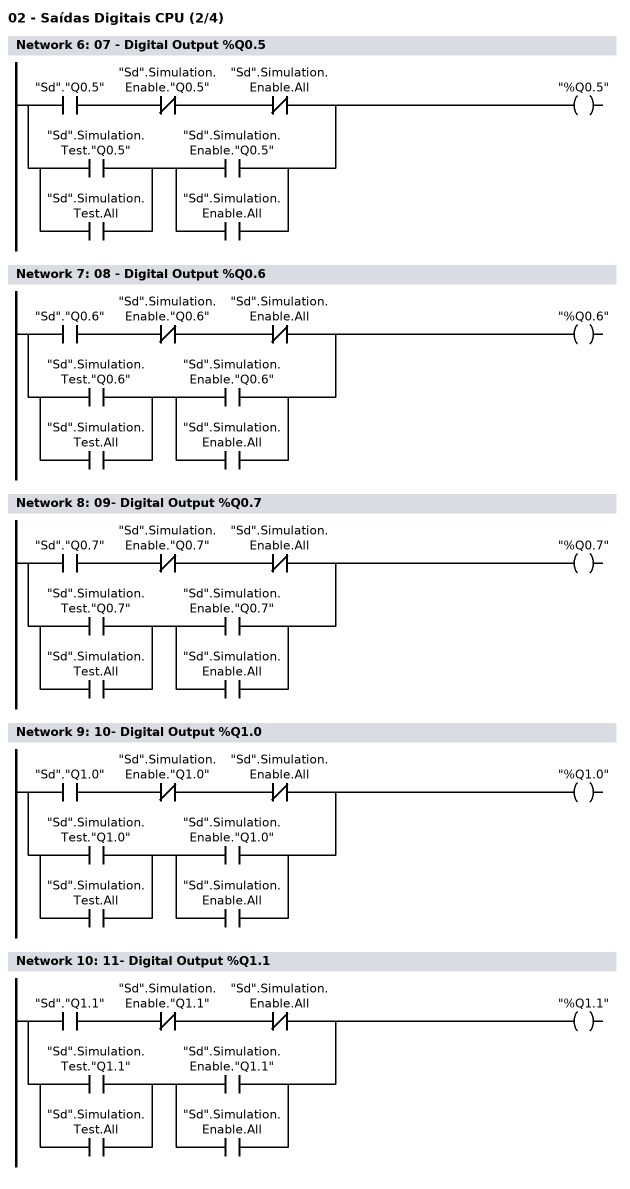
   RUNG wire#powerrail
      Contact( "Sd"."Q0.5" )
      I_Contact( "Sd".Simulation.Enable."Q0.5" )
      I_Contact( "Sd".Simulation.Enable.All )
      wire#w1
      Coil( "%Q0.5" )
   END_RUNG
   RUNG wire#powerrail
      Contact( "Sd".Simulation.Test."Q0.5" )
      wire#w2
      Contact( "Sd".Simulation.Enable."Q0.5" )
   END_RUNG wire#w1
   RUNG wire#powerrail
      Contact( "Sd".Simulation.Test.All )
   END_RUNG wire#w2
   RUNG wire#w2
      Contact( "Sd".Simulation.Enable.All )
   END_RUNG wire#w1
   // the same network as SCL:
   "%Q0.5" := ("Sd"."Q0.5" AND NOT "Sd".Simulation.Enable."Q0.5" AND NOT "Sd".Simulation.Enable.All) OR (("Sd".Simulation.Test."Q0.5" OR "Sd".Simulation.Test.All) AND ("Sd".Simulation.Enable."Q0.5" OR "Sd".Simulation.Enable.All));
END_REGION

REGION Network 7: 08 - Digital Output %Q0.6
   RUNG wire#powerrail
      Contact( "Sd"."Q0.6" )
      I_Contact( "Sd".Simulation.Enable."Q0.6" )
      I_Contact( "Sd".Simulation.Enable.All )
      wire#w1
      Coil( "%Q0.6" )
   END_RUNG
   RUNG wire#powerrail
      Contact( "Sd".Simulation.Test."Q0.6" )
      wire#w2
      Contact( "Sd".Simulation.Enable."Q0.6" )
   END_RUNG wire#w1
   RUNG wire#powerrail
      Contact( "Sd".Simulation.Test.All )
   END_RUNG wire#w2
   RUNG wire#w2
      Contact( "Sd".Simulation.Enable.All )
   END_RUNG wire#w1
   // the same network as SCL:
   "%Q0.6" := ("Sd"."Q0.6" AND NOT "Sd".Simulation.Enable."Q0.6" AND NOT "Sd".Simulation.Enable.All) OR (("Sd".Simulation.Test."Q0.6" OR "Sd".Simulation.Test.All) AND ("Sd".Simulation.Enable."Q0.6" OR "Sd".Simulation.Enable.All));
END_REGION

REGION Network 8: 09- Digital Output %Q0.7
   RUNG wire#powerrail
      Contact( "Sd"."Q0.7" )
      I_Contact( "Sd".Simulation.Enable."Q0.7" )
      I_Contact( "Sd".Simulation.Enable.All )
      wire#w1
      Coil( "%Q0.7" )
   END_RUNG
   RUNG wire#powerrail
      Contact( "Sd".Simulation.Test."Q0.7" )
      wire#w2
      Contact( "Sd".Simulation.Enable."Q0.7" )
   END_RUNG wire#w1
   RUNG wire#powerrail
      Contact( "Sd".Simulation.Test.All )
   END_RUNG wire#w2
   RUNG wire#w2
      Contact( "Sd".Simulation.Enable.All )
   END_RUNG wire#w1
   // the same network as SCL:
   "%Q0.7" := ("Sd"."Q0.7" AND NOT "Sd".Simulation.Enable."Q0.7" AND NOT "Sd".Simulation.Enable.All) OR (("Sd".Simulation.Test."Q0.7" OR "Sd".Simulation.Test.All) AND ("Sd".Simulation.Enable."Q0.7" OR "Sd".Simulation.Enable.All));
END_REGION

REGION Network 9: 10- Digital Output %Q1.0
   RUNG wire#powerrail
      Contact( "Sd"."Q1.0" )
      I_Contact( "Sd".Simulation.Enable."Q1.0" )
      I_Contact( "Sd".Simulation.Enable.All )
      wire#w1
      Coil( "%Q1.0" )
   END_RUNG
   RUNG wire#powerrail
      Contact( "Sd".Simulation.Test."Q1.0" )
      wire#w2
      Contact( "Sd".Simulation.Enable."Q1.0" )
   END_RUNG wire#w1
   RUNG wire#powerrail
      Contact( "Sd".Simulation.Test.All )
   END_RUNG wire#w2
   RUNG wire#w2
      Contact( "Sd".Simulation.Enable.All )
   END_RUNG wire#w1
   // the same network as SCL:
   "%Q1.0" := ("Sd"."Q1.0" AND NOT "Sd".Simulation.Enable."Q1.0" AND NOT "Sd".Simulation.Enable.All) OR (("Sd".Simulation.Test."Q1.0" OR "Sd".Simulation.Test.All) AND ("Sd".Simulation.Enable."Q1.0" OR "Sd".Simulation.Enable.All));
END_REGION

REGION Network 10: 11- Digital Output %Q1.1
   RUNG wire#powerrail
      Contact( "Sd"."Q1.1" )
      I_Contact( "Sd".Simulation.Enable."Q1.1" )
      I_Contact( "Sd".Simulation.Enable.All )
      wire#w1
      Coil( "%Q1.1" )
   END_RUNG
   RUNG wire#powerrail
      Contact( "Sd".Simulation.Test."Q1.1" )
      wire#w2
      Contact( "Sd".Simulation.Enable."Q1.1" )
   END_RUNG wire#w1
   RUNG wire#powerrail
      Contact( "Sd".Simulation.Test.All )
   END_RUNG wire#w2
   RUNG wire#w2
      Contact( "Sd".Simulation.Enable.All )
   END_RUNG wire#w1
   // the same network as SCL:
   "%Q1.1" := ("Sd"."Q1.1" AND NOT "Sd".Simulation.Enable."Q1.1" AND NOT "Sd".Simulation.Enable.All) OR (("Sd".Simulation.Test."Q1.1" OR "Sd".Simulation.Test.All) AND ("Sd".Simulation.Enable."Q1.1" OR "Sd".Simulation.Enable.All));
END_REGION

REGION Network 11: 11- Digital Output %Q1.2
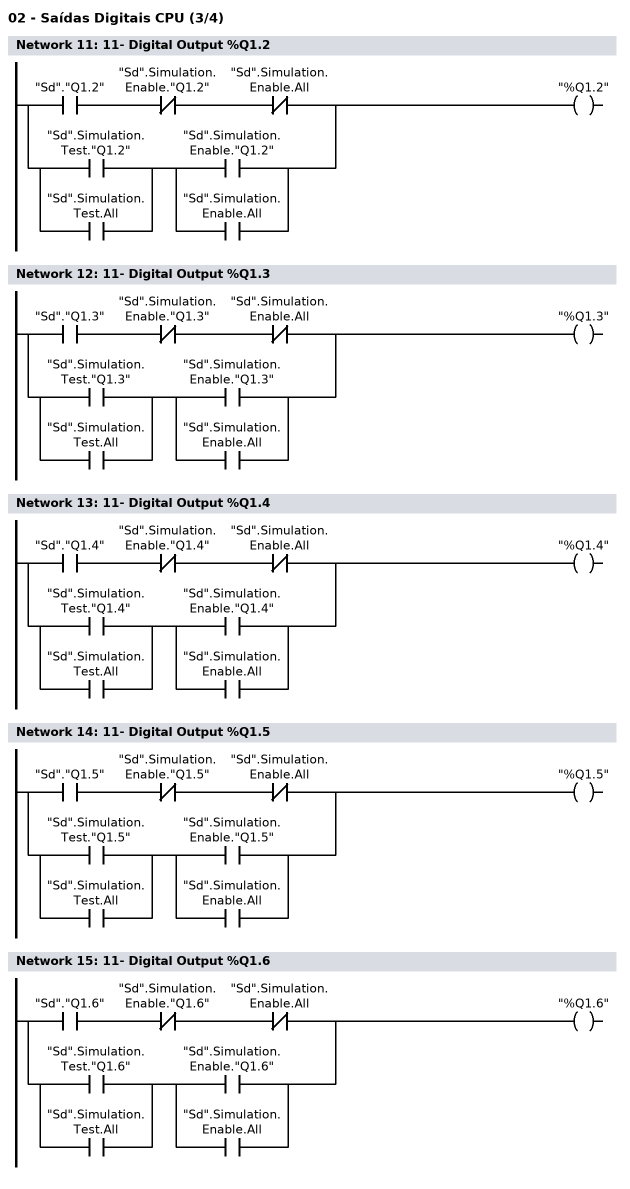
   RUNG wire#powerrail
      Contact( "Sd"."Q1.2" )
      I_Contact( "Sd".Simulation.Enable."Q1.2" )
      I_Contact( "Sd".Simulation.Enable.All )
      wire#w1
      Coil( "%Q1.2" )
   END_RUNG
   RUNG wire#powerrail
      Contact( "Sd".Simulation.Test."Q1.2" )
      wire#w2
      Contact( "Sd".Simulation.Enable."Q1.2" )
   END_RUNG wire#w1
   RUNG wire#powerrail
      Contact( "Sd".Simulation.Test.All )
   END_RUNG wire#w2
   RUNG wire#w2
      Contact( "Sd".Simulation.Enable.All )
   END_RUNG wire#w1
   // the same network as SCL:
   "%Q1.2" := ("Sd"."Q1.2" AND NOT "Sd".Simulation.Enable."Q1.2" AND NOT "Sd".Simulation.Enable.All) OR (("Sd".Simulation.Test."Q1.2" OR "Sd".Simulation.Test.All) AND ("Sd".Simulation.Enable."Q1.2" OR "Sd".Simulation.Enable.All));
END_REGION

REGION Network 12: 11- Digital Output %Q1.3
   RUNG wire#powerrail
      Contact( "Sd"."Q1.3" )
      I_Contact( "Sd".Simulation.Enable."Q1.3" )
      I_Contact( "Sd".Simulation.Enable.All )
      wire#w1
      Coil( "%Q1.3" )
   END_RUNG
   RUNG wire#powerrail
      Contact( "Sd".Simulation.Test."Q1.3" )
      wire#w2
      Contact( "Sd".Simulation.Enable."Q1.3" )
   END_RUNG wire#w1
   RUNG wire#powerrail
      Contact( "Sd".Simulation.Test.All )
   END_RUNG wire#w2
   RUNG wire#w2
      Contact( "Sd".Simulation.Enable.All )
   END_RUNG wire#w1
   // the same network as SCL:
   "%Q1.3" := ("Sd"."Q1.3" AND NOT "Sd".Simulation.Enable."Q1.3" AND NOT "Sd".Simulation.Enable.All) OR (("Sd".Simulation.Test."Q1.3" OR "Sd".Simulation.Test.All) AND ("Sd".Simulation.Enable."Q1.3" OR "Sd".Simulation.Enable.All));
END_REGION

REGION Network 13: 11- Digital Output %Q1.4
   RUNG wire#powerrail
      Contact( "Sd"."Q1.4" )
      I_Contact( "Sd".Simulation.Enable."Q1.4" )
      I_Contact( "Sd".Simulation.Enable.All )
      wire#w1
      Coil( "%Q1.4" )
   END_RUNG
   RUNG wire#powerrail
      Contact( "Sd".Simulation.Test."Q1.4" )
      wire#w2
      Contact( "Sd".Simulation.Enable."Q1.4" )
   END_RUNG wire#w1
   RUNG wire#powerrail
      Contact( "Sd".Simulation.Test.All )
   END_RUNG wire#w2
   RUNG wire#w2
      Contact( "Sd".Simulation.Enable.All )
   END_RUNG wire#w1
   // the same network as SCL:
   "%Q1.4" := ("Sd"."Q1.4" AND NOT "Sd".Simulation.Enable."Q1.4" AND NOT "Sd".Simulation.Enable.All) OR (("Sd".Simulation.Test."Q1.4" OR "Sd".Simulation.Test.All) AND ("Sd".Simulation.Enable."Q1.4" OR "Sd".Simulation.Enable.All));
END_REGION

REGION Network 14: 11- Digital Output %Q1.5
   RUNG wire#powerrail
      Contact( "Sd"."Q1.5" )
      I_Contact( "Sd".Simulation.Enable."Q1.5" )
      I_Contact( "Sd".Simulation.Enable.All )
      wire#w1
      Coil( "%Q1.5" )
   END_RUNG
   RUNG wire#powerrail
      Contact( "Sd".Simulation.Test."Q1.5" )
      wire#w2
      Contact( "Sd".Simulation.Enable."Q1.5" )
   END_RUNG wire#w1
   RUNG wire#powerrail
      Contact( "Sd".Simulation.Test.All )
   END_RUNG wire#w2
   RUNG wire#w2
      Contact( "Sd".Simulation.Enable.All )
   END_RUNG wire#w1
   // the same network as SCL:
   "%Q1.5" := ("Sd"."Q1.5" AND NOT "Sd".Simulation.Enable."Q1.5" AND NOT "Sd".Simulation.Enable.All) OR (("Sd".Simulation.Test."Q1.5" OR "Sd".Simulation.Test.All) AND ("Sd".Simulation.Enable."Q1.5" OR "Sd".Simulation.Enable.All));
END_REGION

REGION Network 15: 11- Digital Output %Q1.6
   RUNG wire#powerrail
      Contact( "Sd"."Q1.6" )
      I_Contact( "Sd".Simulation.Enable."Q1.6" )
      I_Contact( "Sd".Simulation.Enable.All )
      wire#w1
      Coil( "%Q1.6" )
   END_RUNG
   RUNG wire#powerrail
      Contact( "Sd".Simulation.Test."Q1.6" )
      wire#w2
      Contact( "Sd".Simulation.Enable."Q1.6" )
   END_RUNG wire#w1
   RUNG wire#powerrail
      Contact( "Sd".Simulation.Test.All )
   END_RUNG wire#w2
   RUNG wire#w2
      Contact( "Sd".Simulation.Enable.All )
   END_RUNG wire#w1
   // the same network as SCL:
   "%Q1.6" := ("Sd"."Q1.6" AND NOT "Sd".Simulation.Enable."Q1.6" AND NOT "Sd".Simulation.Enable.All) OR (("Sd".Simulation.Test."Q1.6" OR "Sd".Simulation.Test.All) AND ("Sd".Simulation.Enable."Q1.6" OR "Sd".Simulation.Enable.All));
END_REGION

REGION Network 16: 11- Digital Output %Q1.7
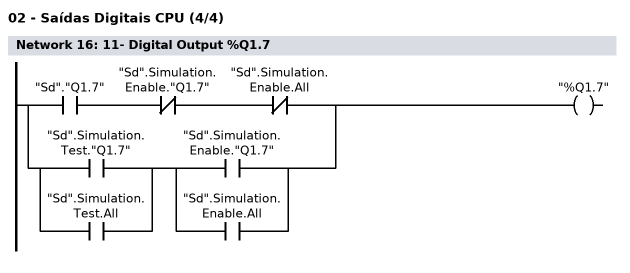
   RUNG wire#powerrail
      Contact( "Sd"."Q1.7" )
      I_Contact( "Sd".Simulation.Enable."Q1.7" )
      I_Contact( "Sd".Simulation.Enable.All )
      wire#w1
      Coil( "%Q1.7" )
   END_RUNG
   RUNG wire#powerrail
      Contact( "Sd".Simulation.Test."Q1.7" )
      wire#w2
      Contact( "Sd".Simulation.Enable."Q1.7" )
   END_RUNG wire#w1
   RUNG wire#powerrail
      Contact( "Sd".Simulation.Test.All )
   END_RUNG wire#w2
   RUNG wire#w2
      Contact( "Sd".Simulation.Enable.All )
   END_RUNG wire#w1
   // the same network as SCL:
   "%Q1.7" := ("Sd"."Q1.7" AND NOT "Sd".Simulation.Enable."Q1.7" AND NOT "Sd".Simulation.Enable.All) OR (("Sd".Simulation.Test."Q1.7" OR "Sd".Simulation.Test.All) AND ("Sd".Simulation.Enable."Q1.7" OR "Sd".Simulation.Enable.All));
END_REGION
END_FUNCTION

FUNCTION "03 - Entradas Analógicas CPU" : Void   // FC3, LAD
TITLE = Analog Inputs
{ S7_Optimized_Access := 'TRUE' }
VERSION : 0.1
// 03 - Analog Inputs
   VAR_TEMP
      TESTE : Int;
   END_VAR
BEGIN

REGION Network 1: Analog Input %IW2 - Limits
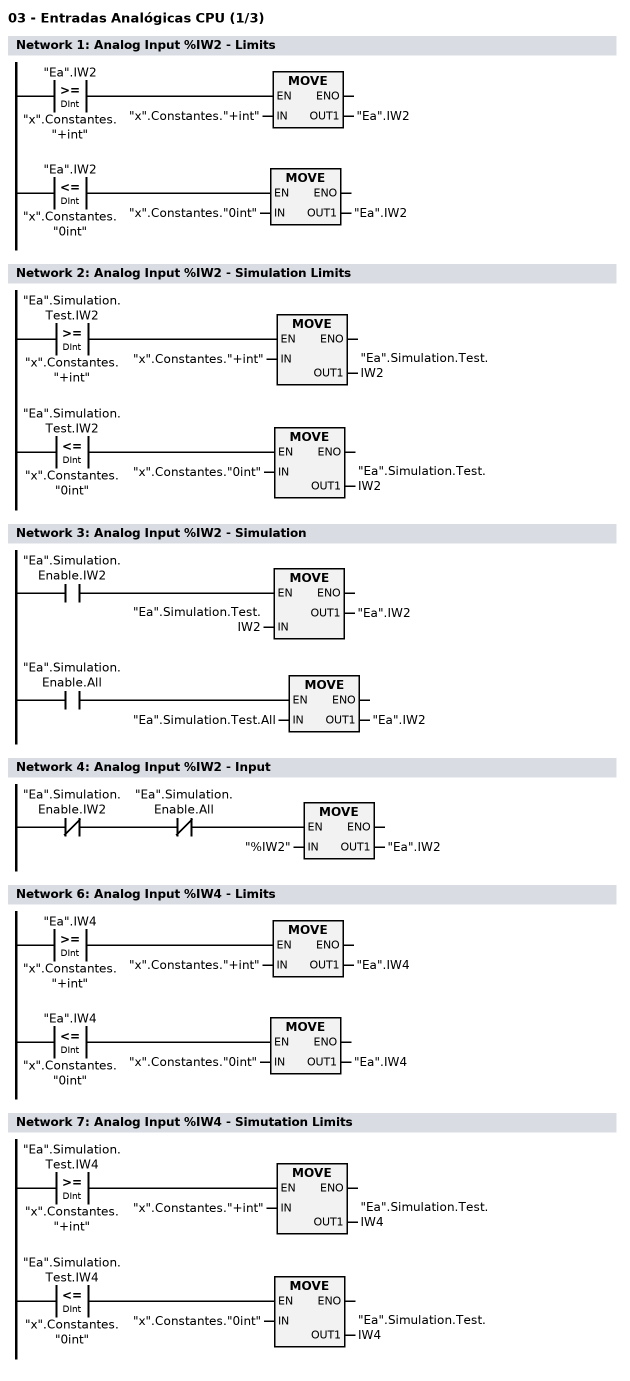
   RUNG wire#powerrail
      { S7_Templates := "SrcType := DInt" } GE_Contact(in1 := "Ea".IW2, in2 := "x".Constantes."+int")
      Move(in := "x".Constantes."+int", out1 => "Ea".IW2)
   END_RUNG
   RUNG wire#powerrail
      { S7_Templates := "SrcType := DInt" } LE_Contact(in1 := "Ea".IW2, in2 := "x".Constantes."0int")
      Move(in := "x".Constantes."0int", out1 => "Ea".IW2)
   END_RUNG
   // the same network as SCL:
   IF "Ea".IW2 >= "x".Constantes."+int" THEN "Ea".IW2 := "x".Constantes."+int"; END_IF;
   IF "Ea".IW2 <= "x".Constantes."0int" THEN "Ea".IW2 := "x".Constantes."0int"; END_IF;
END_REGION

REGION Network 2: Analog Input %IW2 - Simulation Limits
   RUNG wire#powerrail
      { S7_Templates := "SrcType := DInt" } GE_Contact(in1 := "Ea".Simulation.Test.IW2, in2 := "x".Constantes."+int")
      Move(in := "x".Constantes."+int", out1 => "Ea".Simulation.Test.IW2)
   END_RUNG
   RUNG wire#powerrail
      { S7_Templates := "SrcType := DInt" } LE_Contact(in1 := "Ea".Simulation.Test.IW2, in2 := "x".Constantes."0int")
      Move(in := "x".Constantes."0int", out1 => "Ea".Simulation.Test.IW2)
   END_RUNG
   // the same network as SCL:
   IF "Ea".Simulation.Test.IW2 >= "x".Constantes."+int" THEN
       "Ea".Simulation.Test.IW2 := "x".Constantes."+int";
   END_IF;
   IF "Ea".Simulation.Test.IW2 <= "x".Constantes."0int" THEN
       "Ea".Simulation.Test.IW2 := "x".Constantes."0int";
   END_IF;
END_REGION

REGION Network 3: Analog Input %IW2 - Simulation
   RUNG wire#powerrail
      Contact( "Ea".Simulation.Enable.IW2 )
      Move(in := "Ea".Simulation.Test.IW2, out1 => "Ea".IW2)
   END_RUNG
   RUNG wire#powerrail
      Contact( "Ea".Simulation.Enable.All )
      Move(in := "Ea".Simulation.Test.All, out1 => "Ea".IW2)
   END_RUNG
   // the same network as SCL:
   IF "Ea".Simulation.Enable.IW2 THEN "Ea".IW2 := "Ea".Simulation.Test.IW2; END_IF;
   IF "Ea".Simulation.Enable.All THEN "Ea".IW2 := "Ea".Simulation.Test.All; END_IF;
END_REGION

REGION Network 4: Analog Input %IW2 - Input
   RUNG wire#powerrail
      I_Contact( "Ea".Simulation.Enable.IW2 )
      I_Contact( "Ea".Simulation.Enable.All )
      Move(in := "%IW2", out1 => "Ea".IW2)
   END_RUNG
   // the same network as SCL:
   IF NOT "Ea".Simulation.Enable.IW2 AND NOT "Ea".Simulation.Enable.All THEN "Ea".IW2 := "%IW2"; END_IF;
END_REGION

REGION Network 5: ############################
END_REGION

REGION Network 6: Analog Input %IW4 - Limits
   RUNG wire#powerrail
      { S7_Templates := "SrcType := DInt" } GE_Contact(in1 := "Ea".IW4, in2 := "x".Constantes."+int")
      Move(in := "x".Constantes."+int", out1 => "Ea".IW4)
   END_RUNG
   RUNG wire#powerrail
      { S7_Templates := "SrcType := DInt" } LE_Contact(in1 := "Ea".IW4, in2 := "x".Constantes."0int")
      Move(in := "x".Constantes."0int", out1 => "Ea".IW4)
   END_RUNG
   // the same network as SCL:
   IF "Ea".IW4 >= "x".Constantes."+int" THEN "Ea".IW4 := "x".Constantes."+int"; END_IF;
   IF "Ea".IW4 <= "x".Constantes."0int" THEN "Ea".IW4 := "x".Constantes."0int"; END_IF;
END_REGION

REGION Network 7: Analog Input %IW4 - Simutation Limits
   RUNG wire#powerrail
      { S7_Templates := "SrcType := DInt" } GE_Contact(in1 := "Ea".Simulation.Test.IW4, in2 := "x".Constantes."+int")
      Move(in := "x".Constantes."+int", out1 => "Ea".Simulation.Test.IW4)
   END_RUNG
   RUNG wire#powerrail
      { S7_Templates := "SrcType := DInt" } LE_Contact(in1 := "Ea".Simulation.Test.IW4, in2 := "x".Constantes."0int")
      Move(in := "x".Constantes."0int", out1 => "Ea".Simulation.Test.IW4)
   END_RUNG
   // the same network as SCL:
   IF "Ea".Simulation.Test.IW4 >= "x".Constantes."+int" THEN
       "Ea".Simulation.Test.IW4 := "x".Constantes."+int";
   END_IF;
   IF "Ea".Simulation.Test.IW4 <= "x".Constantes."0int" THEN
       "Ea".Simulation.Test.IW4 := "x".Constantes."0int";
   END_IF;
END_REGION

REGION Network 8: Analog Input %IW4 - Simulation
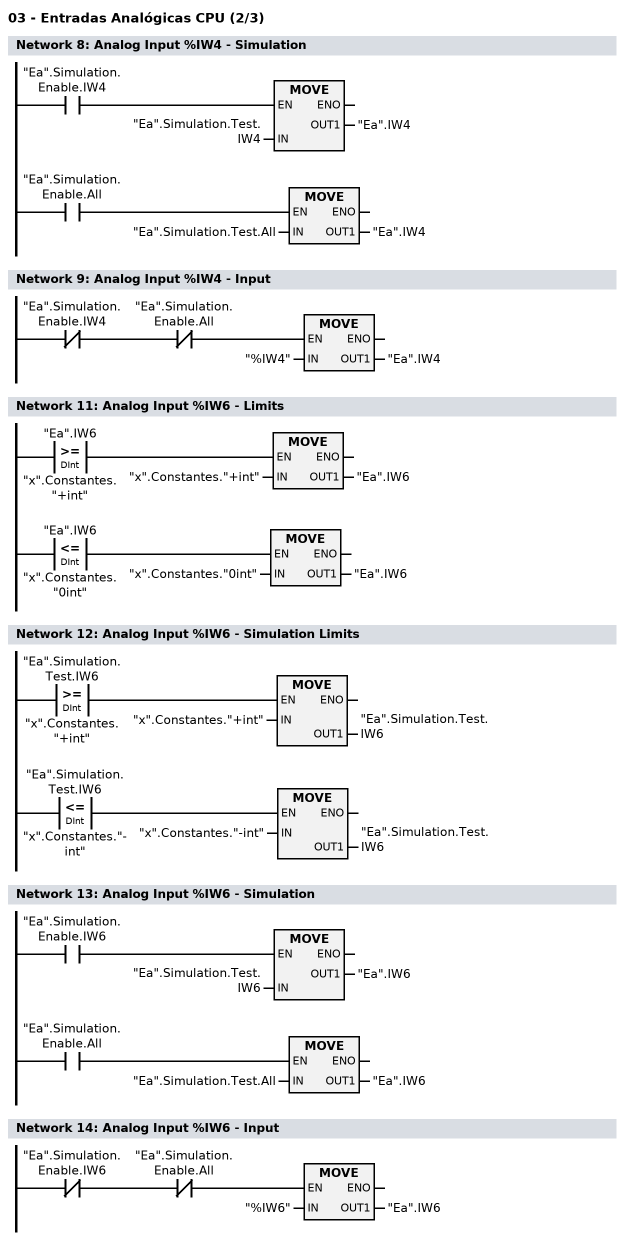
   RUNG wire#powerrail
      Contact( "Ea".Simulation.Enable.IW4 )
      Move(in := "Ea".Simulation.Test.IW4, out1 => "Ea".IW4)
   END_RUNG
   RUNG wire#powerrail
      Contact( "Ea".Simulation.Enable.All )
      Move(in := "Ea".Simulation.Test.All, out1 => "Ea".IW4)
   END_RUNG
   // the same network as SCL:
   IF "Ea".Simulation.Enable.IW4 THEN "Ea".IW4 := "Ea".Simulation.Test.IW4; END_IF;
   IF "Ea".Simulation.Enable.All THEN "Ea".IW4 := "Ea".Simulation.Test.All; END_IF;
END_REGION

REGION Network 9: Analog Input %IW4 - Input
   RUNG wire#powerrail
      I_Contact( "Ea".Simulation.Enable.IW4 )
      I_Contact( "Ea".Simulation.Enable.All )
      Move(in := "%IW4", out1 => "Ea".IW4)
   END_RUNG
   // the same network as SCL:
   IF NOT "Ea".Simulation.Enable.IW4 AND NOT "Ea".Simulation.Enable.All THEN "Ea".IW4 := "%IW4"; END_IF;
END_REGION

REGION Network 10: ############################
END_REGION

REGION Network 11: Analog Input %IW6 - Limits
   RUNG wire#powerrail
      { S7_Templates := "SrcType := DInt" } GE_Contact(in1 := "Ea".IW6, in2 := "x".Constantes."+int")
      Move(in := "x".Constantes."+int", out1 => "Ea".IW6)
   END_RUNG
   RUNG wire#powerrail
      { S7_Templates := "SrcType := DInt" } LE_Contact(in1 := "Ea".IW6, in2 := "x".Constantes."0int")
      Move(in := "x".Constantes."0int", out1 => "Ea".IW6)
   END_RUNG
   // the same network as SCL:
   IF "Ea".IW6 >= "x".Constantes."+int" THEN "Ea".IW6 := "x".Constantes."+int"; END_IF;
   IF "Ea".IW6 <= "x".Constantes."0int" THEN "Ea".IW6 := "x".Constantes."0int"; END_IF;
END_REGION

REGION Network 12: Analog Input %IW6 - Simulation Limits
   RUNG wire#powerrail
      { S7_Templates := "SrcType := DInt" } GE_Contact(in1 := "Ea".Simulation.Test.IW6, in2 := "x".Constantes."+int")
      Move(in := "x".Constantes."+int", out1 => "Ea".Simulation.Test.IW6)
   END_RUNG
   RUNG wire#powerrail
      { S7_Templates := "SrcType := DInt" } LE_Contact(in1 := "Ea".Simulation.Test.IW6, in2 := "x".Constantes."-int")
      Move(in := "x".Constantes."-int", out1 => "Ea".Simulation.Test.IW6)
   END_RUNG
   // the same network as SCL:
   IF "Ea".Simulation.Test.IW6 >= "x".Constantes."+int" THEN
       "Ea".Simulation.Test.IW6 := "x".Constantes."+int";
   END_IF;
   IF "Ea".Simulation.Test.IW6 <= "x".Constantes."-int" THEN
       "Ea".Simulation.Test.IW6 := "x".Constantes."-int";
   END_IF;
END_REGION

REGION Network 13: Analog Input %IW6 - Simulation
   RUNG wire#powerrail
      Contact( "Ea".Simulation.Enable.IW6 )
      Move(in := "Ea".Simulation.Test.IW6, out1 => "Ea".IW6)
   END_RUNG
   RUNG wire#powerrail
      Contact( "Ea".Simulation.Enable.All )
      Move(in := "Ea".Simulation.Test.All, out1 => "Ea".IW6)
   END_RUNG
   // the same network as SCL:
   IF "Ea".Simulation.Enable.IW6 THEN "Ea".IW6 := "Ea".Simulation.Test.IW6; END_IF;
   IF "Ea".Simulation.Enable.All THEN "Ea".IW6 := "Ea".Simulation.Test.All; END_IF;
END_REGION

REGION Network 14: Analog Input %IW6 - Input
   RUNG wire#powerrail
      I_Contact( "Ea".Simulation.Enable.IW6 )
      I_Contact( "Ea".Simulation.Enable.All )
      Move(in := "%IW6", out1 => "Ea".IW6)
   END_RUNG
   // the same network as SCL:
   IF NOT "Ea".Simulation.Enable.IW6 AND NOT "Ea".Simulation.Enable.All THEN "Ea".IW6 := "%IW6"; END_IF;
END_REGION

REGION Network 15: ############################
END_REGION

REGION Network 16: Analog Input %IW8 - Limits
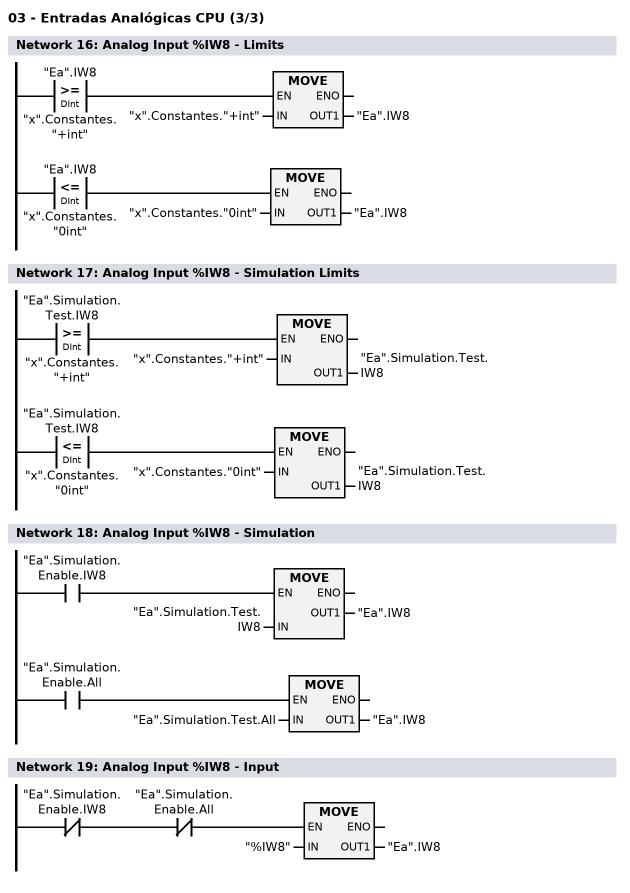
   RUNG wire#powerrail
      { S7_Templates := "SrcType := DInt" } GE_Contact(in1 := "Ea".IW8, in2 := "x".Constantes."+int")
      Move(in := "x".Constantes."+int", out1 => "Ea".IW8)
   END_RUNG
   RUNG wire#powerrail
      { S7_Templates := "SrcType := DInt" } LE_Contact(in1 := "Ea".IW8, in2 := "x".Constantes."0int")
      Move(in := "x".Constantes."0int", out1 => "Ea".IW8)
   END_RUNG
   // the same network as SCL:
   IF "Ea".IW8 >= "x".Constantes."+int" THEN "Ea".IW8 := "x".Constantes."+int"; END_IF;
   IF "Ea".IW8 <= "x".Constantes."0int" THEN "Ea".IW8 := "x".Constantes."0int"; END_IF;
END_REGION

REGION Network 17: Analog Input %IW8 - Simulation Limits
   RUNG wire#powerrail
      { S7_Templates := "SrcType := DInt" } GE_Contact(in1 := "Ea".Simulation.Test.IW8, in2 := "x".Constantes."+int")
      Move(in := "x".Constantes."+int", out1 => "Ea".Simulation.Test.IW8)
   END_RUNG
   RUNG wire#powerrail
      { S7_Templates := "SrcType := DInt" } LE_Contact(in1 := "Ea".Simulation.Test.IW8, in2 := "x".Constantes."0int")
      Move(in := "x".Constantes."0int", out1 => "Ea".Simulation.Test.IW8)
   END_RUNG
   // the same network as SCL:
   IF "Ea".Simulation.Test.IW8 >= "x".Constantes."+int" THEN
       "Ea".Simulation.Test.IW8 := "x".Constantes."+int";
   END_IF;
   IF "Ea".Simulation.Test.IW8 <= "x".Constantes."0int" THEN
       "Ea".Simulation.Test.IW8 := "x".Constantes."0int";
   END_IF;
END_REGION

REGION Network 18: Analog Input %IW8 - Simulation
   RUNG wire#powerrail
      Contact( "Ea".Simulation.Enable.IW8 )
      Move(in := "Ea".Simulation.Test.IW8, out1 => "Ea".IW8)
   END_RUNG
   RUNG wire#powerrail
      Contact( "Ea".Simulation.Enable.All )
      Move(in := "Ea".Simulation.Test.All, out1 => "Ea".IW8)
   END_RUNG
   // the same network as SCL:
   IF "Ea".Simulation.Enable.IW8 THEN "Ea".IW8 := "Ea".Simulation.Test.IW8; END_IF;
   IF "Ea".Simulation.Enable.All THEN "Ea".IW8 := "Ea".Simulation.Test.All; END_IF;
END_REGION

REGION Network 19: Analog Input %IW8 - Input
   RUNG wire#powerrail
      I_Contact( "Ea".Simulation.Enable.IW8 )
      I_Contact( "Ea".Simulation.Enable.All )
      Move(in := "%IW8", out1 => "Ea".IW8)
   END_RUNG
   // the same network as SCL:
   IF NOT "Ea".Simulation.Enable.IW8 AND NOT "Ea".Simulation.Enable.All THEN "Ea".IW8 := "%IW8"; END_IF;
END_REGION
END_FUNCTION

FUNCTION "04 - Saídas Analógicas CPU" : Void   // FC4, LAD
TITLE = 04 - Analog Outputs
{ S7_Optimized_Access := 'TRUE' }
VERSION : 0.1
// 04 - Analog Outputs
BEGIN

REGION Network 1: Analog Output %QW2 - Limits
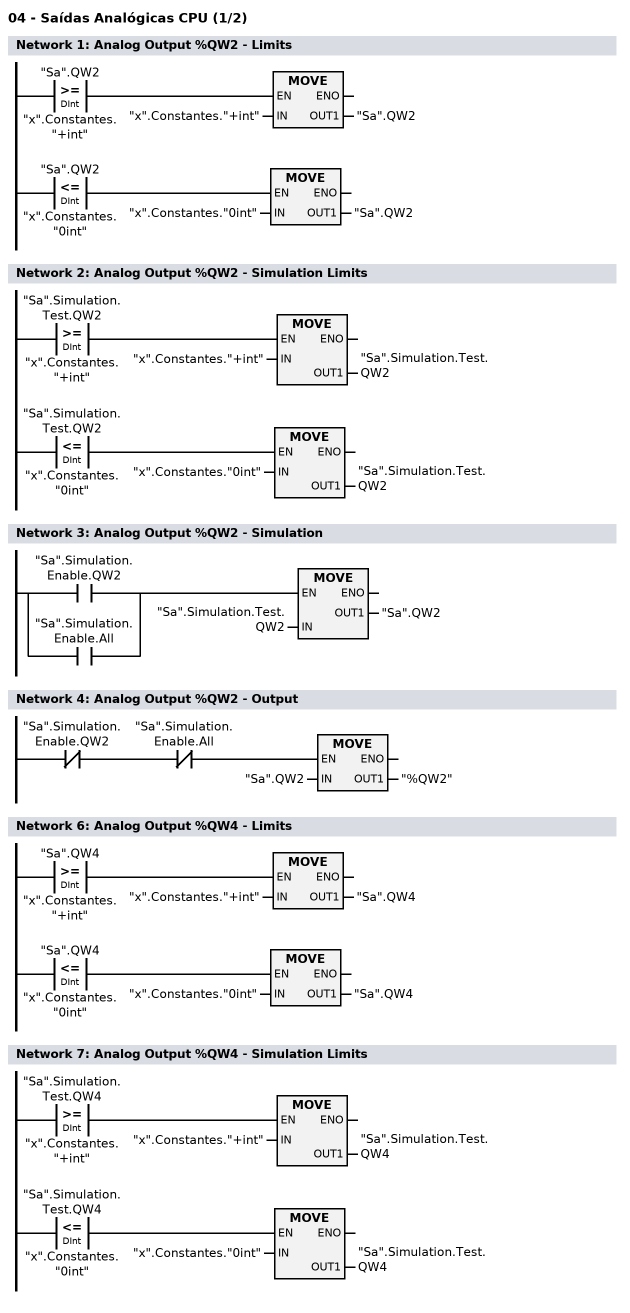
   RUNG wire#powerrail
      { S7_Templates := "SrcType := DInt" } GE_Contact(in1 := "Sa".QW2, in2 := "x".Constantes."+int")
      Move(in := "x".Constantes."+int", out1 => "Sa".QW2)
   END_RUNG
   RUNG wire#powerrail
      { S7_Templates := "SrcType := DInt" } LE_Contact(in1 := "Sa".QW2, in2 := "x".Constantes."0int")
      Move(in := "x".Constantes."0int", out1 => "Sa".QW2)
   END_RUNG
   // the same network as SCL:
   IF "Sa".QW2 >= "x".Constantes."+int" THEN "Sa".QW2 := "x".Constantes."+int"; END_IF;
   IF "Sa".QW2 <= "x".Constantes."0int" THEN "Sa".QW2 := "x".Constantes."0int"; END_IF;
END_REGION

REGION Network 2: Analog Output %QW2 - Simulation Limits
   RUNG wire#powerrail
      { S7_Templates := "SrcType := DInt" } GE_Contact(in1 := "Sa".Simulation.Test.QW2, in2 := "x".Constantes."+int")
      Move(in := "x".Constantes."+int", out1 => "Sa".Simulation.Test.QW2)
   END_RUNG
   RUNG wire#powerrail
      { S7_Templates := "SrcType := DInt" } LE_Contact(in1 := "Sa".Simulation.Test.QW2, in2 := "x".Constantes."0int")
      Move(in := "x".Constantes."0int", out1 => "Sa".Simulation.Test.QW2)
   END_RUNG
   // the same network as SCL:
   IF "Sa".Simulation.Test.QW2 >= "x".Constantes."+int" THEN
       "Sa".Simulation.Test.QW2 := "x".Constantes."+int";
   END_IF;
   IF "Sa".Simulation.Test.QW2 <= "x".Constantes."0int" THEN
       "Sa".Simulation.Test.QW2 := "x".Constantes."0int";
   END_IF;
END_REGION

REGION Network 3: Analog Output %QW2 - Simulation
   RUNG wire#powerrail
      Contact( "Sa".Simulation.Enable.QW2 )
      wire#w1
      Move(in := "Sa".Simulation.Test.QW2, out1 => "Sa".QW2)
   END_RUNG
   RUNG wire#powerrail
      Contact( "Sa".Simulation.Enable.All )
   END_RUNG wire#w1
   // the same network as SCL:
   IF "Sa".Simulation.Enable.QW2 OR "Sa".Simulation.Enable.All THEN
       "Sa".QW2 := "Sa".Simulation.Test.QW2;
   END_IF;
END_REGION

REGION Network 4: Analog Output %QW2 - Output
   RUNG wire#powerrail
      I_Contact( "Sa".Simulation.Enable.QW2 )
      I_Contact( "Sa".Simulation.Enable.All )
      Move(in := "Sa".QW2, out1 => "%QW2")
   END_RUNG
   // the same network as SCL:
   IF NOT "Sa".Simulation.Enable.QW2 AND NOT "Sa".Simulation.Enable.All THEN "%QW2" := "Sa".QW2; END_IF;
END_REGION

REGION Network 5: ##################################
END_REGION

REGION Network 6: Analog Output %QW4 - Limits
   RUNG wire#powerrail
      { S7_Templates := "SrcType := DInt" } GE_Contact(in1 := "Sa".QW4, in2 := "x".Constantes."+int")
      Move(in := "x".Constantes."+int", out1 => "Sa".QW4)
   END_RUNG
   RUNG wire#powerrail
      { S7_Templates := "SrcType := DInt" } LE_Contact(in1 := "Sa".QW4, in2 := "x".Constantes."0int")
      Move(in := "x".Constantes."0int", out1 => "Sa".QW4)
   END_RUNG
   // the same network as SCL:
   IF "Sa".QW4 >= "x".Constantes."+int" THEN "Sa".QW4 := "x".Constantes."+int"; END_IF;
   IF "Sa".QW4 <= "x".Constantes."0int" THEN "Sa".QW4 := "x".Constantes."0int"; END_IF;
END_REGION

REGION Network 7: Analog Output %QW4 - Simulation Limits
   RUNG wire#powerrail
      { S7_Templates := "SrcType := DInt" } GE_Contact(in1 := "Sa".Simulation.Test.QW4, in2 := "x".Constantes."+int")
      Move(in := "x".Constantes."+int", out1 => "Sa".Simulation.Test.QW4)
   END_RUNG
   RUNG wire#powerrail
      { S7_Templates := "SrcType := DInt" } LE_Contact(in1 := "Sa".Simulation.Test.QW4, in2 := "x".Constantes."0int")
      Move(in := "x".Constantes."0int", out1 => "Sa".Simulation.Test.QW4)
   END_RUNG
   // the same network as SCL:
   IF "Sa".Simulation.Test.QW4 >= "x".Constantes."+int" THEN
       "Sa".Simulation.Test.QW4 := "x".Constantes."+int";
   END_IF;
   IF "Sa".Simulation.Test.QW4 <= "x".Constantes."0int" THEN
       "Sa".Simulation.Test.QW4 := "x".Constantes."0int";
   END_IF;
END_REGION

REGION Network 8: Analog Output %QW4 - Simulation
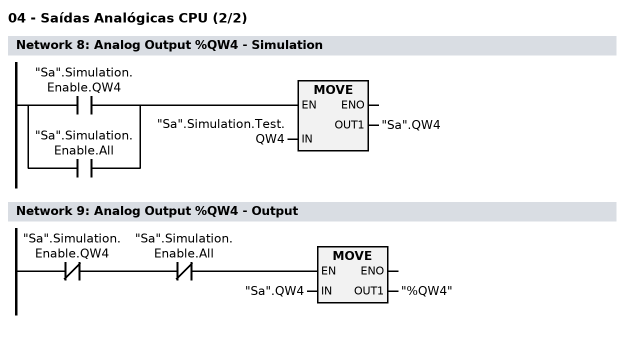
   RUNG wire#powerrail
      Contact( "Sa".Simulation.Enable.QW4 )
      wire#w1
      Move(in := "Sa".Simulation.Test.QW4, out1 => "Sa".QW4)
   END_RUNG
   RUNG wire#powerrail
      Contact( "Sa".Simulation.Enable.All )
   END_RUNG wire#w1
   // the same network as SCL:
   IF "Sa".Simulation.Enable.QW4 OR "Sa".Simulation.Enable.All THEN
       "Sa".QW4 := "Sa".Simulation.Test.QW4;
   END_IF;
END_REGION

REGION Network 9: Analog Output %QW4 - Output
   RUNG wire#powerrail
      I_Contact( "Sa".Simulation.Enable.QW4 )
      I_Contact( "Sa".Simulation.Enable.All )
      Move(in := "Sa".QW4, out1 => "%QW4")
   END_RUNG
   // the same network as SCL:
   IF NOT "Sa".Simulation.Enable.QW4 AND NOT "Sa".Simulation.Enable.All THEN "%QW4" := "Sa".QW4; END_IF;
END_REGION
END_FUNCTION

// folder: 002 - Comunication Node-Red

FUNCTION "01 - Node-Red" : Void   // FC5, LAD
{ S7_Optimized_Access := 'TRUE' }
VERSION : 0.1
   VAR_TEMP
      auxWriteNodRedReal : Real;
   END_VAR
   VAR_TEMP   // added for the SCL form of the ladder/FBD networks
      _w1 : Bool;
      _w2 : Bool;
   END_VAR
BEGIN

REGION Network 1: Recebe Valor Bool Node-Red
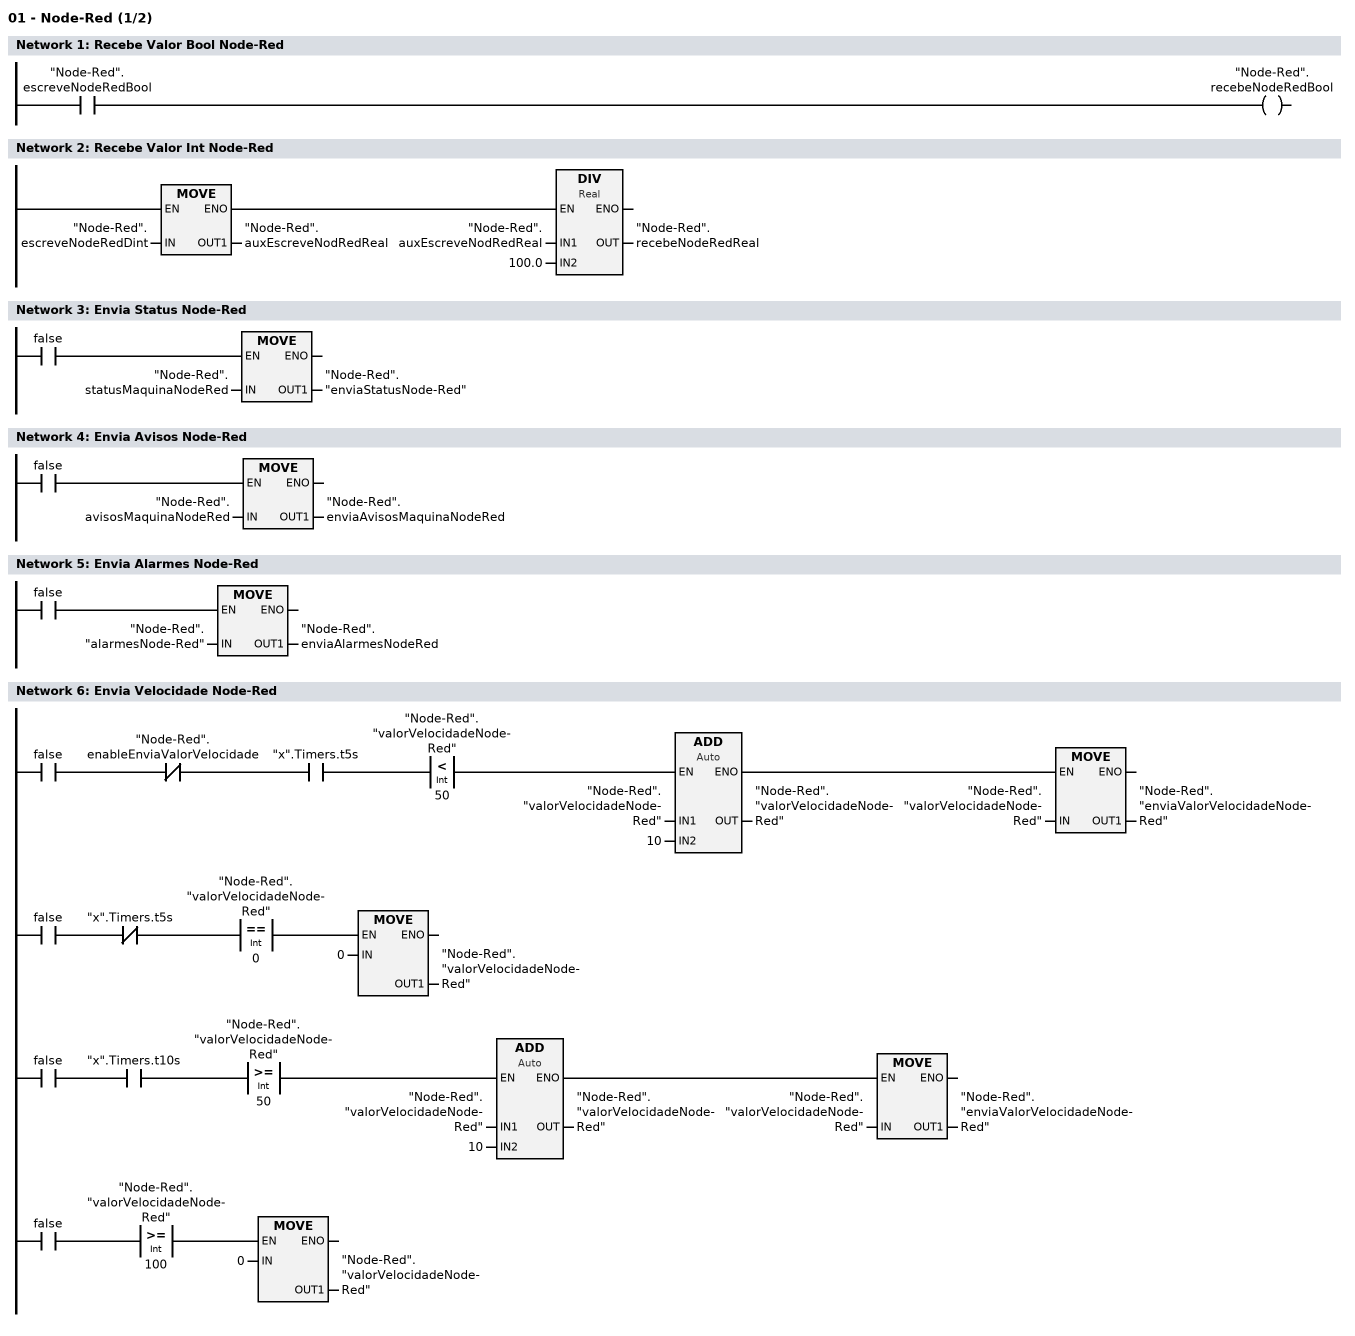
   RUNG wire#powerrail
      Contact( "Node-Red".escreveNodeRedBool )
      Coil( "Node-Red".recebeNodeRedBool )
   END_RUNG
   // the same network as SCL:
   "Node-Red".recebeNodeRedBool := "Node-Red".escreveNodeRedBool;
END_REGION

REGION Network 2: Recebe Valor Int Node-Red
   RUNG wire#powerrail
      Move(in := "Node-Red".escreveNodeRedDint, out1 => "Node-Red".auxEscreveNodRedReal)
      { S7_Templates := "SrcType := Real" } Div(in1 := "Node-Red".auxEscreveNodRedReal, in2 := 100.0, out => "Node-Red".recebeNodeRedReal)
   END_RUNG
   // the same network as SCL:
   "Node-Red".auxEscreveNodRedReal := "Node-Red".escreveNodeRedDint;
   "Node-Red".recebeNodeRedReal := "Node-Red".auxEscreveNodRedReal / 100.0;
END_REGION

REGION Network 3: Envia Status Node-Red
   RUNG wire#powerrail
      Contact( false )
      Move(in := "Node-Red".statusMaquinaNodeRed, out1 => "Node-Red"."enviaStatusNode-Red")
   END_RUNG
   // the same network as SCL:
   IF false THEN "Node-Red"."enviaStatusNode-Red" := "Node-Red".statusMaquinaNodeRed; END_IF;
END_REGION

REGION Network 4: Envia Avisos Node-Red
   RUNG wire#powerrail
      Contact( false )
      Move(in := "Node-Red".avisosMaquinaNodeRed, out1 => "Node-Red".enviaAvisosMaquinaNodeRed)
   END_RUNG
   // the same network as SCL:
   IF false THEN "Node-Red".enviaAvisosMaquinaNodeRed := "Node-Red".avisosMaquinaNodeRed; END_IF;
END_REGION

REGION Network 5: Envia Alarmes Node-Red
   RUNG wire#powerrail
      Contact( false )
      Move(in := "Node-Red"."alarmesNode-Red", out1 => "Node-Red".enviaAlarmesNodeRed)
   END_RUNG
   // the same network as SCL:
   IF false THEN "Node-Red".enviaAlarmesNodeRed := "Node-Red"."alarmesNode-Red"; END_IF;
END_REGION

REGION Network 6: Envia Velocidade Node-Red
   RUNG wire#powerrail
      Contact( false )
      I_Contact( "Node-Red".enableEnviaValorVelocidade )
      Contact( "x".Timers.t5s )
      { S7_Templates := "SrcType := Int" } LT_Contact(in1 := "Node-Red"."valorVelocidadeNode-Red", in2 := 50)
      Add(in1 := "Node-Red"."valorVelocidadeNode-Red", in2 := 10, out => "Node-Red"."valorVelocidadeNode-Red")
      Move(in := "Node-Red"."valorVelocidadeNode-Red", out1 => "Node-Red"."enviaValorVelocidadeNode-Red")
   END_RUNG
   RUNG wire#powerrail
      Contact( false )
      I_Contact( "x".Timers.t5s )
      { S7_Templates := "SrcType := Int" } EQ_Contact(in1 := "Node-Red"."valorVelocidadeNode-Red", in2 := 0)
      Move(in := 0, out1 => "Node-Red"."valorVelocidadeNode-Red")
   END_RUNG
   RUNG wire#powerrail
      Contact( false )
      Contact( "x".Timers.t10s )
      { S7_Templates := "SrcType := Int" } GE_Contact(in1 := "Node-Red"."valorVelocidadeNode-Red", in2 := 50)
      Add(in1 := "Node-Red"."valorVelocidadeNode-Red", in2 := 10, out => "Node-Red"."valorVelocidadeNode-Red")
      Move(in := "Node-Red"."valorVelocidadeNode-Red", out1 => "Node-Red"."enviaValorVelocidadeNode-Red")
   END_RUNG
   RUNG wire#powerrail
      Contact( false )
      { S7_Templates := "SrcType := Int" } GE_Contact(in1 := "Node-Red"."valorVelocidadeNode-Red", in2 := 100)
      Move(in := 0, out1 => "Node-Red"."valorVelocidadeNode-Red")
   END_RUNG
   // the same network as SCL:
   #_w1 := false AND NOT "Node-Red".enableEnviaValorVelocidade AND "x".Timers.t5s AND ("Node-Red"."valorVelocidadeNode-Red" < 50);
   IF #_w1 THEN
       "Node-Red"."valorVelocidadeNode-Red" := "Node-Red"."valorVelocidadeNode-Red" + 10;
       "Node-Red"."enviaValorVelocidadeNode-Red" := "Node-Red"."valorVelocidadeNode-Red";
   END_IF;
   IF false AND NOT "x".Timers.t5s AND ("Node-Red"."valorVelocidadeNode-Red" = 0) THEN
       "Node-Red"."valorVelocidadeNode-Red" := 0;
   END_IF;
   #_w2 := false AND "x".Timers.t10s AND ("Node-Red"."valorVelocidadeNode-Red" >= 50);
   IF #_w2 THEN
       "Node-Red"."valorVelocidadeNode-Red" := "Node-Red"."valorVelocidadeNode-Red" + 10;
       "Node-Red"."enviaValorVelocidadeNode-Red" := "Node-Red"."valorVelocidadeNode-Red";
   END_IF;
   IF false AND ("Node-Red"."valorVelocidadeNode-Red" >= 100) THEN
       "Node-Red"."valorVelocidadeNode-Red" := 0;
   END_IF;
END_REGION

REGION Network 7: Envia Valor de Produção
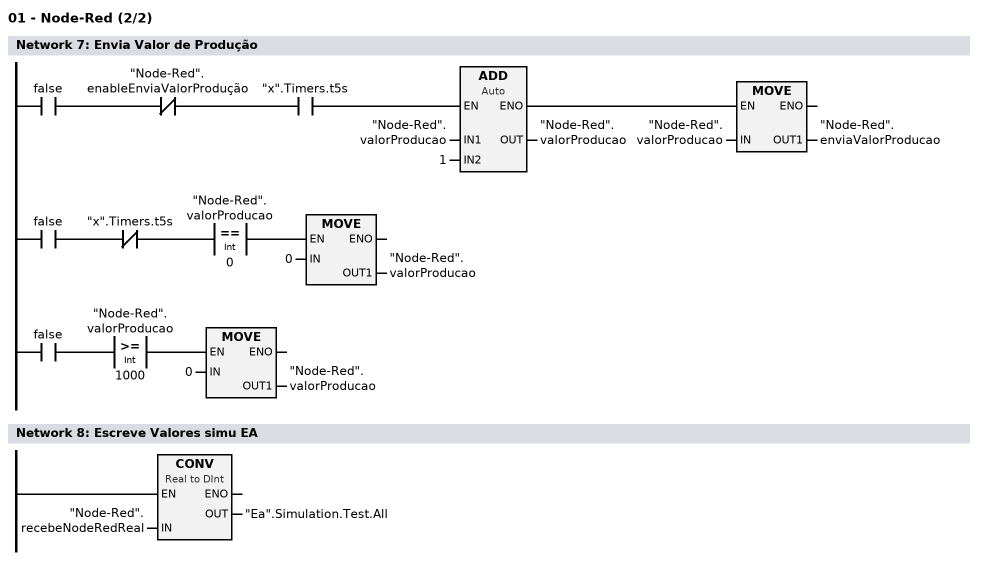
   RUNG wire#powerrail
      Contact( false )
      I_Contact( "Node-Red".enableEnviaValorProdução )
      Contact( "x".Timers.t5s )
      Add(in1 := "Node-Red".valorProducao, in2 := 1, out => "Node-Red".valorProducao)
      Move(in := "Node-Red".valorProducao, out1 => "Node-Red".enviaValorProducao)
   END_RUNG
   RUNG wire#powerrail
      Contact( false )
      I_Contact( "x".Timers.t5s )
      { S7_Templates := "SrcType := Int" } EQ_Contact(in1 := "Node-Red".valorProducao, in2 := 0)
      Move(in := 0, out1 => "Node-Red".valorProducao)
   END_RUNG
   RUNG wire#powerrail
      Contact( false )
      { S7_Templates := "SrcType := Int" } GE_Contact(in1 := "Node-Red".valorProducao, in2 := 1000)
      Move(in := 0, out1 => "Node-Red".valorProducao)
   END_RUNG
   // the same network as SCL:
   IF false AND NOT "Node-Red".enableEnviaValorProdução AND "x".Timers.t5s THEN
       "Node-Red".valorProducao := "Node-Red".valorProducao + 1;
       "Node-Red".enviaValorProducao := "Node-Red".valorProducao;
   END_IF;
   IF false AND NOT "x".Timers.t5s AND ("Node-Red".valorProducao = 0) THEN
       "Node-Red".valorProducao := 0;
   END_IF;
   IF false AND ("Node-Red".valorProducao >= 1000) THEN "Node-Red".valorProducao := 0; END_IF;
END_REGION

REGION Network 8: Escreve Valores simu EA
   RUNG wire#powerrail
      { S7_Templates := "[SrcType := Real, DestType := DInt]" } Convert(in := "Node-Red".recebeNodeRedReal, out => "Ea".Simulation.Test.All)
   END_RUNG
   // the same network as SCL:
   "Ea".Simulation.Test.All := REAL_TO_DINT("Node-Red".recebeNodeRedReal);
END_REGION
END_FUNCTION

FUNCTION "02 - Alarmes" : Void   // FC6, LAD
TITLE = Envio de Alarmes da Máquina para Node-RED
{ S7_Optimized_Access := 'TRUE' }
VERSION : 0.1
BEGIN

REGION Network 1: Envio de Alarmes da Máquina para Node-RED
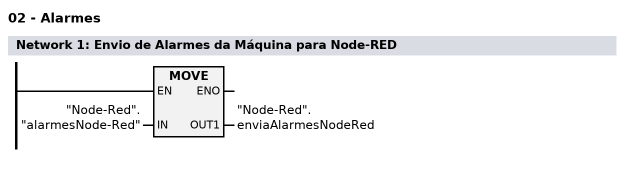
   RUNG wire#powerrail
      Move(in := "Node-Red"."alarmesNode-Red", out1 => "Node-Red".enviaAlarmesNodeRed)
   END_RUNG
   // the same network as SCL:
   "Node-Red".enviaAlarmesNodeRed := "Node-Red"."alarmesNode-Red";
END_REGION
END_FUNCTION

FUNCTION "03 - Avisos" : Void   // FC7, LAD
TITLE = Envio de Aviso da Máquina para Node-RED
{ S7_Optimized_Access := 'TRUE' }
VERSION : 0.1
BEGIN

REGION Network 1: Envio de Aviso da Máquina para Node-RED
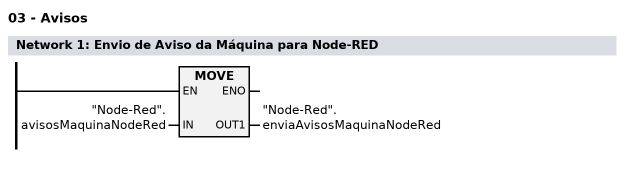
   RUNG wire#powerrail
      Move(in := "Node-Red".avisosMaquinaNodeRed, out1 => "Node-Red".enviaAvisosMaquinaNodeRed)
   END_RUNG
   // the same network as SCL:
   "Node-Red".enviaAvisosMaquinaNodeRed := "Node-Red".avisosMaquinaNodeRed;
END_REGION
END_FUNCTION

FUNCTION "04 - Status" : Void   // FC8, LAD
TITLE = Envio de Status da Máquina para Node-RED
{ S7_Optimized_Access := 'TRUE' }
VERSION : 0.1
BEGIN

REGION Network 1: Envio de Status da Máquina para Node-RED
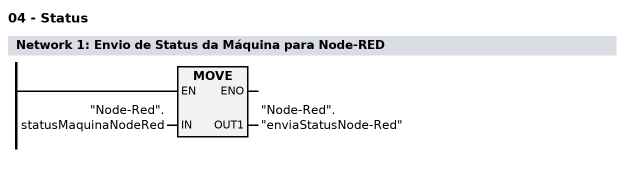
   RUNG wire#powerrail
      Move(in := "Node-Red".statusMaquinaNodeRed, out1 => "Node-Red"."enviaStatusNode-Red")
   END_RUNG
   // the same network as SCL:
   "Node-Red"."enviaStatusNode-Red" := "Node-Red".statusMaquinaNodeRed;
END_REGION
END_FUNCTION

FUNCTION "05 - Velocidade" : Void   // FC9, LAD
TITLE = Envio de Velocidade da Máquina para Node-RED
{ S7_Optimized_Access := 'TRUE' }
VERSION : 0.1
   VAR_TEMP   // added for the SCL form of the ladder/FBD networks
      _w1 : Bool;
      _w2 : Bool;
   END_VAR
BEGIN

REGION Network 1: Envio de Velocidade da Máquina para Node-RED
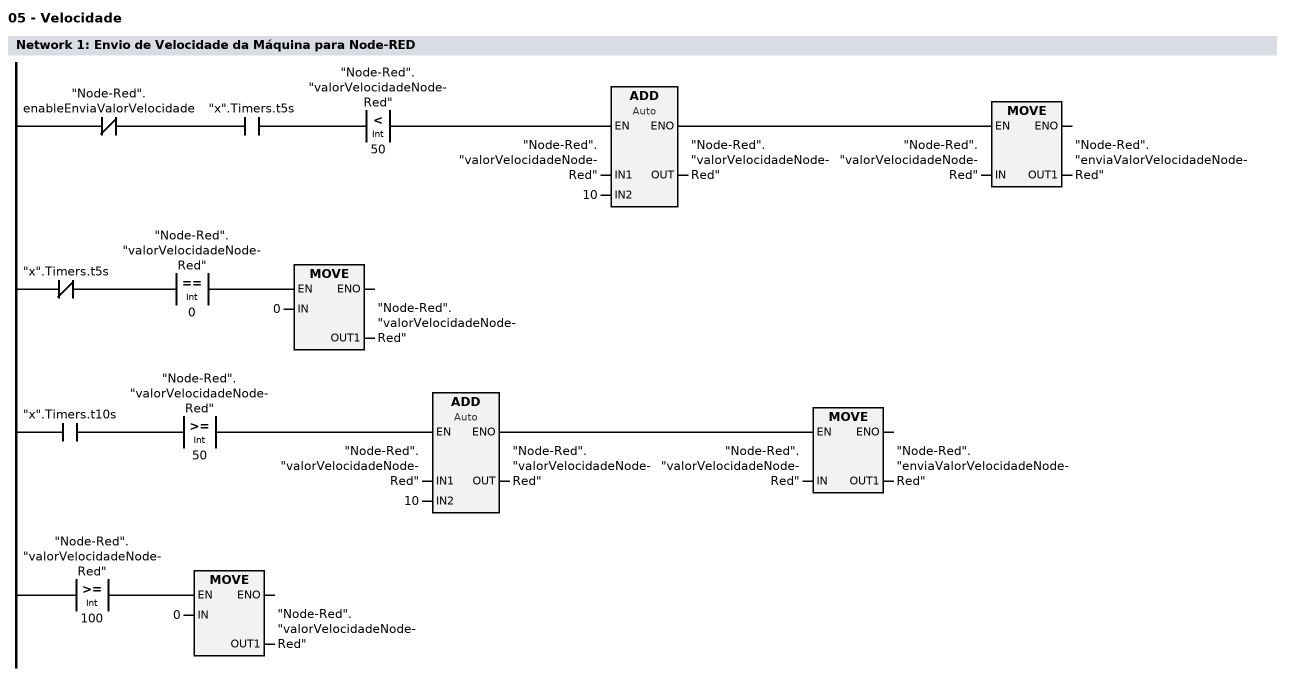
   RUNG wire#powerrail
      I_Contact( "Node-Red".enableEnviaValorVelocidade )
      Contact( "x".Timers.t5s )
      { S7_Templates := "SrcType := Int" } LT_Contact(in1 := "Node-Red"."valorVelocidadeNode-Red", in2 := 50)
      Add(in1 := "Node-Red"."valorVelocidadeNode-Red", in2 := 10, out => "Node-Red"."valorVelocidadeNode-Red")
      Move(in := "Node-Red"."valorVelocidadeNode-Red", out1 => "Node-Red"."enviaValorVelocidadeNode-Red")
   END_RUNG
   RUNG wire#powerrail
      I_Contact( "x".Timers.t5s )
      { S7_Templates := "SrcType := Int" } EQ_Contact(in1 := "Node-Red"."valorVelocidadeNode-Red", in2 := 0)
      Move(in := 0, out1 => "Node-Red"."valorVelocidadeNode-Red")
   END_RUNG
   RUNG wire#powerrail
      Contact( "x".Timers.t10s )
      { S7_Templates := "SrcType := Int" } GE_Contact(in1 := "Node-Red"."valorVelocidadeNode-Red", in2 := 50)
      Add(in1 := "Node-Red"."valorVelocidadeNode-Red", in2 := 10, out => "Node-Red"."valorVelocidadeNode-Red")
      Move(in := "Node-Red"."valorVelocidadeNode-Red", out1 => "Node-Red"."enviaValorVelocidadeNode-Red")
   END_RUNG
   RUNG wire#powerrail
      { S7_Templates := "SrcType := Int" } GE_Contact(in1 := "Node-Red"."valorVelocidadeNode-Red", in2 := 100)
      Move(in := 0, out1 => "Node-Red"."valorVelocidadeNode-Red")
   END_RUNG
   // the same network as SCL:
   #_w1 := NOT "Node-Red".enableEnviaValorVelocidade AND "x".Timers.t5s AND ("Node-Red"."valorVelocidadeNode-Red" < 50);
   IF #_w1 THEN
       "Node-Red"."valorVelocidadeNode-Red" := "Node-Red"."valorVelocidadeNode-Red" + 10;
       "Node-Red"."enviaValorVelocidadeNode-Red" := "Node-Red"."valorVelocidadeNode-Red";
   END_IF;
   IF NOT "x".Timers.t5s AND ("Node-Red"."valorVelocidadeNode-Red" = 0) THEN
       "Node-Red"."valorVelocidadeNode-Red" := 0;
   END_IF;
   #_w2 := "x".Timers.t10s AND ("Node-Red"."valorVelocidadeNode-Red" >= 50);
   IF #_w2 THEN
       "Node-Red"."valorVelocidadeNode-Red" := "Node-Red"."valorVelocidadeNode-Red" + 10;
       "Node-Red"."enviaValorVelocidadeNode-Red" := "Node-Red"."valorVelocidadeNode-Red";
   END_IF;
   IF "Node-Red"."valorVelocidadeNode-Red" >= 100 THEN "Node-Red"."valorVelocidadeNode-Red" := 0; END_IF;
END_REGION
END_FUNCTION

FUNCTION "06 - Produção" : Void   // FC10, LAD
TITLE = Envio de Produção da Máquina para Node-RED
{ S7_Optimized_Access := 'TRUE' }
VERSION : 0.1
BEGIN

REGION Network 1: Envio de Produção da Máquina para Node-RED
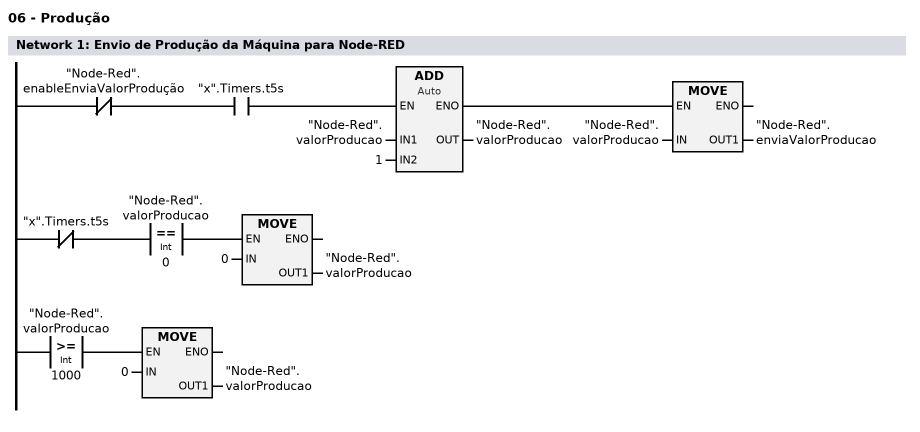
   RUNG wire#powerrail
      I_Contact( "Node-Red".enableEnviaValorProdução )
      Contact( "x".Timers.t5s )
      Add(in1 := "Node-Red".valorProducao, in2 := 1, out => "Node-Red".valorProducao)
      Move(in := "Node-Red".valorProducao, out1 => "Node-Red".enviaValorProducao)
   END_RUNG
   RUNG wire#powerrail
      I_Contact( "x".Timers.t5s )
      { S7_Templates := "SrcType := Int" } EQ_Contact(in1 := "Node-Red".valorProducao, in2 := 0)
      Move(in := 0, out1 => "Node-Red".valorProducao)
   END_RUNG
   RUNG wire#powerrail
      { S7_Templates := "SrcType := Int" } GE_Contact(in1 := "Node-Red".valorProducao, in2 := 1000)
      Move(in := 0, out1 => "Node-Red".valorProducao)
   END_RUNG
   // the same network as SCL:
   IF NOT "Node-Red".enableEnviaValorProdução AND "x".Timers.t5s THEN
       "Node-Red".valorProducao := "Node-Red".valorProducao + 1;
       "Node-Red".enviaValorProducao := "Node-Red".valorProducao;
   END_IF;
   IF NOT "x".Timers.t5s AND ("Node-Red".valorProducao = 0) THEN "Node-Red".valorProducao := 0; END_IF;
   IF "Node-Red".valorProducao >= 1000 THEN "Node-Red".valorProducao := 0; END_IF;
END_REGION
END_FUNCTION